VAR_INPUT
	WatchDog	: BOOL;
	// I/O Inputs 
		//FROM ENEDIS
		IN_CmdAutCpl_IO							: BOOL; 			(* Coupling Authorization (Autorisation de couplage)			              	*)
		IN_CmdAutCpl_End_IO						: BOOL; 			(* End of coupling Authorization (Fin d'autorisation de couplage)			    *)
		IN_CmdDisconnect_End_IO					: BOOL; 			(* End of disconnect order(Fin de demande de decouplage)                        *)
		IN_CmdDisconnect_IO						: BOOL;				(* Disconnect order(Demande de decouplage)                                      *)
		IN_CmdRSEOn_IO							: BOOL;				(* Start of RSE (Mise en RSE)                                                   *)
		IN_CmdRSEOff_IO							: BOOL;				(* Stop of RSE (Mise Hors RSE)                                                  *)
		IN_CmdStopPReg_IO						: BOOL;				(* Desactivation of P0 regulation(Fin de passage a P0)                          *)
		IN_CmdStartPReg_IO						: BOOL;				(* Activation of P0 regulation (Passage a P0)                                   *)
		IN_CmdStopQReg_IO						: BOOL;				(* Desactivation of Q0 regulation(Fin de passage a Q0)                          *)
		IN_CmdStartQreg_IO						: BOOL;				(* Activation of Q0 regulation(Passage a Q0)                                    *)
		IN_CmdEmergencyDisconnect_End_IO		: BOOL;				(* End of Emergency disconnect order(Fin demande d'effacement d'urgence) 	   	*)
		IN_CmdEmergencyDisconnect_IO			: BOOL;				(* Emergency disconnect order(Demande d'effacement d'urgence)                   *)
		IN_CmdDisconnectFromTac_IO				: BOOL; 			(* Teleaction disconnect(Decouplage par tac)                                    *)
		IN_CmdSynchro_IO						: BOOL;				(* Synchronisation signal														*)
		
		(* 4..20mA *)                                   			
		IN_MesP0Reg_IO							: INT; 				(* (kW)   Grid P0	*)
		IN_MesQ0Reg_IO							: INT; 				(* (KVar) Grid Q0 	*)
		IN_MesU0Reg_IO							: INT; 				(* (KV)   Grid V0   *)
		                                                			                                  			
		//FROM AKSES                                    			
		IN_CmdAutCpl_other						: BOOL; 			
		IN_CmdEmergencyDisconnect_other			: BOOL; 			
		IN_CmdEmergencyDisconnect_End_other		: BOOL; 			
		IN_CmdDisconnect_other					: BOOL; 			
		IN_CmdDisconnect_end_other				: BOOL; 			
		IN_CmdStartPReg_other					: BOOL; 			
		IN_CmdStartQReg_other					: BOOL; 			
		IN_CmdStopPReg_other					: BOOL; 			
		IN_CmdStopQReg_other					: BOOL;

		//FROM TAC 
		IN_CmdTAOn_IO							: BOOL; 			(* Teleaction in service(Teleaction en service)                                 *)
		IN_CmdTAOff_IO							: BOOL; 			(* Teleaction out of service (Teleaction Hors service)                          *)
		IN_CmdTacInFault_IO						: BOOL; 			(* Teleaction in fault(Défaut Tac)							 					*)
		IN_CmdOpenTAC_IO						: BOOL; 
		IN_CmdConsignationTAC_IO				: BOOL; 
		IN_CmdUnavailableTAC					: BOOL; 
			
		                                                			
		(*TC Relais Protection*)                        			
		IN_ConnectAuthorizationLost				: BOOL; 			// Tous les cas pour un Reset aut Couplage recu
		IN_Unavailable							: BOOL; 			// Disjoncteur général en Local, ou tous les départs en Local ou Bouton d'arret d'urgence 
		IN_PP_Connected							: BOOL; 			// Centrale Couplée si DG = Fermé et au moins 1 départ antenne en production et au moins un onduleur en Prod
                                     			
		OUT_MesFaultDecoupling_IO				: BOOL; 			(* Decoupling due to faults c13100 and c15400 combined with CB position    	*)
                                             			
END_VAR                                                 			
                                                        			
                                                        			
VAR_OUTPUT 

	// DEIE                                              			
		OUT_MesPPUnavailable_IO					: BOOL; 			(* TS centrale indisponible                                                	*)
		OUT_MesPPConnected_IO					: BOOL; 			(* Centrale couplée(1)/Centrale Découplée(0)                               	*)
		OUT_MesPPDisconnected_IO				: BOOL; 			(* Centrale Découplée														*)
		OUT_MesAutCpl_IO 						: BOOL; 			(* Autorisation de couplage reçue(1)/Attente d'autorisation de couplage(0)	*)
		OUT_MesAutCpl_end_IO 					: BOOL; 			(* Autorisation de couplage attente                                        	*)
		OUT_MesDisconnect_IO 					: BOOL; 			(* Demande de découplage reçue(1)/Fin de demande de découplage(0)         	*)
		OUT_MesDisconnect_End_IO 				: BOOL; 			(* Demande de découplage attente                                           	*)
		OUT_MesEmergencyDisconnect_IO 			: BOOL; 			(* Demande d effacement d'urgence reçue                                   	*)
		OUT_MesEmergencyDisconnect_End_IO 		: BOOL; 			(* Demande d effacement d'urgence attente		                          	*)
		OUT_MesRSEON_IO							: BOOL; 			(* Demande mise en RSE reçue                                              	*)
		OUT_MesRSEOff_IO						: BOOL; 			(* Demande mise en RSE en attente                                         	*)
		OUT_MesStartPReg_IO						: BOOL; 			(* Demande mise en regulation de P reçue                                  	*)
		OUT_MesStopPReg_IO						: BOOL; 			(* Demande mise en regulation de P en attente                             	*)
		OUT_MesStartQReg_IO						: BOOL; 			(* Demande mise en regulation de Q reçue                                  	*)
		OUT_MesStopQReg_IO						: BOOL; 			(* Demande mise en regulation de Q en attente	                          	*)
		
		(* 4..20mA *)                                   			
		OUT_MesP_IO							: REAL; 				(* (kW)   Grid P0	*)
		OUT_MesQ_IO							: REAL; 				(* (KVar) Grid Q0 	*)
		OUT_MesU_IO							: REAL; 				(* (KV)   Grid V0   *)
		
	// Synchro temporelle - EMS 
		Ecart_HeureGrid						: DINT;
		
	// TAC
		OUT_CmdTacInFault_IO					: BOOL; 
		OUT_MesOpenTAC_IO 						: BOOL; 
		OUT_MesTAOn_IO							: BOOL; 			(* Demande mise en TeleAction reçue                                       	*)
		OUT_MesTAOff_IO							: BOOL; 			(* Demande mise en TeleAction en attente                                  	*)
		
				
	// SOFREL
		
		OUT_MesP_IO_SOFREL					: REAL; 				(* (kW)   Grid P0	*)
		OUT_MesQ_IO_SOFREL					: REAL; 				(* (KVar) Grid Q0 	*)
		OUT_MesU_IO_SOFREL					: REAL; 				(* (KV)   Grid V0   *)
END_VAR


VAR PERSISTENT
	
END_VAR
VAR
		//TON
		TONConnectAuthorization					: TON;
		TONConnectAuthorization_end				: TON;
		TONEmergencyDisconnect	               	: TON;
	    TONEmergencyDisconnect_end	            : TON;
	    TONDisconnect	                		: TON;
	    TONDisconnect_end                		: TON;
	    TONPRegOn				                : TON;
	    TONPRegOff				                : TON;
	    TONQregOn				                : TON;
	    TONQRegOff				                : TON;
	    TONRSEOn				                : TON;
	    TONRSEOff				                : TON;
	    TONTAOn					                : TON;
	    TONTAOff				                : TON;
	
		R_Trig_SynchTime						: R_TRIG;

		Reste 									: DINT;
		Modulo 									: DINT;
		Heure_Pulse 							: DINT;
		bTest 									: BOOL;
END_VAR

METHOD M_AlarmManagement
//////////////////
// alarm and warning management
/////////////////

VAR 
	FB_AlarmCodeManager			: FB_AlarmCodeManager ; 
	
END_VAR
// ALARM CODE //
	FB_AlarmCodeManager(
		bAlarm1			:=MesDataExd.MesData.OUT_MesPPUnavailable, // Power plant is unavailable
		bAlarm2			:=FALSE, //
		bAlarm3			:=FALSE, //
		bAlarm4			:=FALSE, //
		bAlarm5			:=FALSE, //
		bAlarm6			:=FALSE, //
		bAlarm7			:=FALSE, //
		bAlarm8			:=FALSE, //
		bAlarm9			:=FALSE, //
		bAlarm10		:=FALSE, //
		bAlarm11		:=FALSE, //
		bAlarm12		:=FALSE, //
		bAlarm13		:=FALSE, //
		bAlarm14		:=FALSE, //
		bAlarm15		:=FALSE, //						 
		wAlarmCode		=>MesDataExd.MesData.MesAlarmCode);

// WARNING CODE //
	FB_AlarmCodeManager(		
		bAlarm1			:=IN_ConnectAuthorizationLost, 							//Loss of coupling authorization
		bAlarm2			:=FALSE,													//			
		bAlarm3			:=MesDataExd.MesData.OUT_SetptP > ParamPmaxPark OR MesDataExd.MesData.OUT_SetptP <= 0 ,		// P Setpoint from grid outside of permitted range
		bAlarm4			:=MesDataExd.MesData.OUT_SetptQ > ParamQMax OR MesDataExd.MesData.OUT_SetptQ <= ParamQMin, 	// Q Setpoint from grid outside of permitted range
		bAlarm5			:=MesDataExd.MesData.OUT_MesPPConnected						, 	//Powerplant is connected  
		bAlarm6			:=NOT MesDataExd.MesData.OUT_MesPPConnected					, 	//Powerplant is disconnected
		bAlarm7			:=MesDataExd.OUT_CmdPReg							    , 	//Q regulation mode is active     
		bAlarm8			:=NOT MesDataExd.MesData.OUT_CmdAutCpl		    		, 	//Waiting for coupling authorization	
		bAlarm9			:=MesDataExd.MesData.OUT_CmdDisconnect				, 	//Disconnect order
		bAlarm10		:=MesDataExd.MesData.OUT_CmdEmergencyDisconnect 	        , 	//Emergency Disconnect order
		bAlarm11		:=MesDataExd.OUT_CmdPReg												, 	// P regulation mode is active
		bAlarm12		:=MesDataExd.OUT_Rse								    , 	// RSE mode active  
		bAlarm13		:=MesDataExd.OUT_TA 							, 	//Teleaction active
		bAlarm14		:=IN_CmdDisconnectFromTac_IO , 		// Disconnect order from TAC
		bAlarm15		:=IN_CmdTacInFault_IO , 			// TAC in Fault 
		wAlarmCode		=>MesDataExd.MesData.MesWarningCode);		

// EVENT CODE 1//
	FB_AlarmCodeManager(
		bAlarm1			:=FALSE , // 
		bAlarm2			:=NOT MesDataExd.OUT_CmdPReg							    , 	//P regulation mode is inactive
		bAlarm3			:=MesDataExd.MesData.OUT_CmdAutCpl					, 	//Coupling authorization
		bAlarm4			:=FALSE ,//
		bAlarm5			:=IN_CmdSynchro_IO			    						, 	// Synchronization signal 
		bAlarm6			:=NOT MesDataExd.MesData.OUT_CmdDisconnect			, 	//End of disconnect order 
		bAlarm7			:=FALSE ,// 
		bAlarm8			:=NOT MesDataExd.MesData.OUT_CmdEmergencyDisconnect					, 	//End of Emergency Disconnect order
		bAlarm9			:=FALSE , // 
		bAlarm10		:=FALSE , // 
		bAlarm11		:=NOT MesDataExd.OUT_CmdPReg												, 	//P regulation mode is inactive
		bAlarm12		:=FALSE ,//  
		bAlarm13		:=NOT MesDataExd.OUT_Rse							    , 	//RSE mode inactive  
		bAlarm14		:=FALSE ,//
		bAlarm15		:=NOT MesDataExd.OUT_TA							, 	//Teleaction inactive
		wAlarmCode		=>MesDataExd.MesData.MesEventCode);   
                          	
// EVENT CODE 2 //		                                              	
	FB_AlarmCodeManager(                                              	
		bAlarm1			:=IN_CmdAutCpl_IO , 							// Coupling authorization received from DEIE
		bAlarm2			:=IN_CmdDisconnect_End_IO,						// End of disconnect order received from  DEIE
		bAlarm3			:=IN_CmdDisconnect_IO		   , 				// Disconnect order received from DEIE
		bAlarm4			:= IN_CmdEmergencyDisconnect_End_IO	   	, 		// End of Emergency disconnect order received from DEIE
		bAlarm5			:=IN_CmdAutCpl_other, 							// Coupling authoriztion received from HMI
		bAlarm6			:=IN_CmdDisconnect_other		 , 				// Disconnect order received from HMI
		bAlarm7			:=IN_CmdDisconnect_end_other,	 				// End of disconnect order received from HMI
		bAlarm8			:=IN_CmdEmergencyDisconnect_IO	, 				// Emergency disconnect order received from DEIE
		bAlarm9			:=IN_Unavailable, 								// Power plant is unavaiblable ( MainMVCB in local or ES) 
		bAlarm10		:=IN_CmdEmergencyDisconnect_other, 	//Emergency disconnect order received from HMI
		bAlarm11		:=IN_CmdEmergencyDisconnect_End_other	, 	//End of Emergency disconnect order received from HMI
		bAlarm12		:=FALSE, 	//
		bAlarm13		:=FALSE, 	//       
		bAlarm14		:=FALSE, 	//
		bAlarm15		:=FALSE	,//
		wAlarmCode		=>MesDataExd.MesData.MesEventCode2);
END_METHOD

METHOD M_CP
//////////////////
//  Emulator
/////////////////

VAR 
	// Method local variables (reinitialized at each cycle) 
	
END_VAR
END_METHOD

METHOD M_Evaluate
//////////////////
//  Evaluate grid variables 
/////////////////
VAR 
	// Method local variables (reinitialized at each cycle) 
	WatchDog	: BOOL;
END_VAR
WatchDog		:= TRUE;

//Filtering Input
	TONConnectAuthorization		(IN:=IN_CmdAutCpl_IO,PT:=ParamTONFiltering);
	TONEmergencyDisconnect		(IN:=IN_CmdEmergencyDisconnect_IO,PT:=ParamTONFiltering);	
	TONEmergencyDisconnect_end	(IN:=IN_CmdEmergencyDisconnect_End_IO,PT:=ParamTONFiltering);	
	TONDisconnect				(IN:=IN_CmdDisconnect_IO,PT:=ParamTONFiltering);	
	TONDisconnect_end			(IN:=IN_CmdDisconnect_End_IO,PT:=ParamTONFiltering);
	TONPRegOn				(IN:=IN_CmdStartPReg_IO,PT:=ParamTONFiltering);			
	TONPRegOff				(IN:=IN_CmdStopPReg_IO,PT:=ParamTONFiltering);				
	TONQregOn				(IN:=IN_CmdStartQreg_IO,PT:=ParamTONFiltering);				
	TONQRegOff				(IN:=IN_CmdStopQReg_IO,PT:=ParamTONFiltering);				
	TONRSEOn				(IN:=IN_CmdRSEOn_IO,PT:=ParamTONFiltering);				
	TONRSEOff				(IN:=IN_CmdRSEOff_IO,PT:=ParamTONFiltering);				
	TONTAOn					(IN:=IN_CmdTAOn_IO,PT:=ParamTONFiltering);					
	TONTAOff				(IN:=IN_CmdTAOff_IO,PT:=ParamTONFiltering);		

//Filtering Input
	TONConnectAuthorization		(IN:=IN_CmdAutCpl_IO,PT:=ParamTONFiltering);
	TONEmergencyDisconnect		(IN:=IN_CmdEmergencyDisconnect_IO,PT:=ParamTONFiltering);	
	TONEmergencyDisconnect_end	(IN:=IN_CmdEmergencyDisconnect_End_IO,PT:=ParamTONFiltering);	
	TONDisconnect				(IN:=IN_CmdDisconnect_IO,PT:=ParamTONFiltering);	
	TONDisconnect_end			(IN:=IN_CmdDisconnect_End_IO,PT:=ParamTONFiltering);
	TONPRegOn					(IN:=IN_CmdStartPReg_IO,PT:=ParamTONFiltering);			
	TONPRegOff					(IN:=IN_CmdStopPReg_IO,PT:=ParamTONFiltering);				
	TONQregOn					(IN:=IN_CmdStartQreg_IO,PT:=ParamTONFiltering);				
	TONQRegOff					(IN:=IN_CmdStopQReg_IO,PT:=ParamTONFiltering);				
	TONRSEOn					(IN:=IN_CmdRSEOn_IO,PT:=ParamTONFiltering);				
	TONRSEOff					(IN:=IN_CmdRSEOff_IO,PT:=ParamTONFiltering);				
	TONTAOn						(IN:=IN_CmdTAOn_IO,PT:=ParamTONFiltering);					
	TONTAOff					(IN:=IN_CmdTAOff_IO,PT:=ParamTONFiltering);	

// Calculate the difference between the closest hour and the trigger from GRID
	// closest hour is min betwenn the rest of the Euclydian division 3600s = 1h	
	R_Trig_SynchTime(CLK := IN_CmdSynchro_IO OR bTest);
	IF R_Trig_SynchTime.Q THEN
		Heure_Pulse	:= DT_TO_DINT(systemtime_to_dt(TIMESTR := CalLocalTimeStruct));
		Reste := Heure_Pulse MOD 3600;
		IF (3600-Reste) < Reste THEN
			Ecart_HeureGrid := -(3600-Reste);
		ELSE
			Ecart_HeureGrid := Reste;
		END_IF
		//Ecart_HeureGrid := MIN(3600-Reste, Reste);
		MesDataExd.MesEcart_HeureGrid := Ecart_HeureGrid;
	END_IF

//Converting P0 & Q0
	IF ParamP0Available THEN
		//OUT_P0 :=  (MesP0RegIO/ 32767.0) * REAL_TO_INT(ParamPmaxPark);
	MesDataExd.MesData.OUT_SetptP :=  (IN_MesP0Reg_IO/ 32767.0) * ABS(ParamPMin - ParamPmaxPark) + (ParamPMin);
	END_IF
	IF ParamQ0Available THEN
	MesDataExd.MesData.OUT_SetptQ := ( IN_MesQ0Reg_IO / 32767.0) * ABS(ParamQMin - ParamQMax) + (ParamQMin);
	END_IF	
//Logical Equation
	(*PLCUnavailable Si Watchdog n'est pas mis a jour a chaque temps de cycle Ou que la centrale est en Local *)
	MesDataExd.MesData.OUT_MesPPUnavailable := NOT WatchDog OR IN_Unavailable;
	
	(*Centrale Couplée *)
	MesDataExd.MesData.OUT_MesPPConnected := IN_PP_Connected;
	
	(*Autorisation de couplage*)
		IF TONConnectAuthorization.Q OR IN_CmdAutCpl_other THEN
		MesDataExd.MesData.OUT_CmdAutCpl := 1 ;
		END_IF
		
	(*Défaut GTE > 50s : Reset Aut Couplage recus*)
	(*Défaut C13_100 : Reset Aut Couplage recus*)
		IF IN_ConnectAuthorizationLost THEN  //IN_Long_GTE_Fault OR IN_C13_100_Fault OR IN_UnknownFault OR IN_3GTE_Fault THEN
		MesDataExd.MesData.OUT_CmdAutCpl  := FALSE ;
		END_IF
	
	(* RESEAU 6 ET 7 - DEMANDE DE DECOUPLAGE*)
		IF TONDisconnect.Q OR IN_CmdDisconnect_other THEN
			MesDataExd.MesData.OUT_CmdDisconnect := 1 ;
		END_IF
	
		IF TONDisconnect_end.Q OR IN_CmdDisconnect_end_other THEN
		MesDataExd.MesData.OUT_CmdDisconnect := 0 ;
		END_IF

	(* RESEAU 8 ET 9 - DEMANDE D’EFFACEMENT D’URGENCE*)
		IF TONEmergencyDisconnect.Q OR  IN_CmdEmergencyDisconnect_other THEN
		MesDataExd.MesData.OUT_CmdEmergencyDisconnect := 1 ;
		END_IF
	
		IF TONEmergencyDisconnect_end.Q OR IN_CmdEmergencyDisconnect_End_other THEN
		MesDataExd.MesData.OUT_CmdEmergencyDisconnect := 0 ;
		END_IF
	(* RESEAU 10 ET 11 - PASSAGE A P0*)
		IF TONPRegOn.Q OR IN_CmdStartPReg_other THEN
		MesDataExd.OUT_CmdPReg := 1 ;
		END_IF
		
		IF TONPRegOff.Q OR IN_CmdStopPReg_other THEN
		MesDataExd.OUT_CmdPReg := 0 ;
		END_IF
		
	(* RESEAU 12 ET 13 - PASSAGE A Q0*)
		IF TONQregOn.Q OR IN_CmdStartQReg_other THEN
		MesDataExd.OUT_CmdQReg := 1 ;
		END_IF
		
		IF TONQregOff.Q OR IN_CmdStopQReg_other THEN
		MesDataExd.OUT_CmdQReg := 0 ;
		END_IF

				
	(* RSE*)
		IF TONRSEOn.Q  THEN
		MesDataExd.OUT_Rse := 1 ;
		ELSIF TONRSEOff.Q THEN
		MesDataExd.OUT_Rse := 0 ;
		END_IF
		
	(* TA*)
		IF TONTAOn.Q  THEN
		MesDataExd.OUT_TA := 1 ;
		ELSIF TONTAOff.Q THEN
		MesDataExd.OUT_TA := 0 ;
		END_IF
		
	
// Update Outputs IO to GRID 
OUT_MesPPUnavailable_IO				:= MesDataExd.MesData.OUT_MesPPUnavailable ; 			
OUT_MesPPConnected_IO				:= MesDataExd.MesData.OUT_MesPPConnected ; 	
OUT_MesPPDisconnected_IO			:= NOT MesDataExd.MesData.OUT_MesPPConnected ; 
OUT_MesAutCpl_IO 					:= MesDataExd.MesData.OUT_CmdAutCpl ; 			
OUT_MesAutCpl_end_IO 				:= NOT MesDataExd.MesData.OUT_CmdAutCpl ; 		
OUT_MesDisconnect_IO 				:= MesDataExd.MesData.OUT_CmdDisconnect ; 		
OUT_MesDisconnect_End_IO 			:= NOT MesDataExd.MesData.OUT_CmdDisconnect ; 		
OUT_MesEmergencyDisconnect_IO 		:= MesDataExd.MesData.OUT_CmdEmergencyDisconnect ; 		
OUT_MesEmergencyDisconnect_End_IO 	:= NOT MesDataExd.MesData.OUT_CmdEmergencyDisconnect ; 		

OUT_MesRSEON_IO						:= MesDataExd.OUT_Rse ;
OUT_MesRSEOff_IO					:= NOT MesDataExd.OUT_Rse ;
OUT_MesTAOn_IO						:= MesDataExd.OUT_TA ; 
OUT_MesTAOff_IO						:= NOT MesDataExd.OUT_TA ; 

OUT_MesStartPReg_IO	 := MesDataExd.OUT_CmdPReg ; 
OUT_MesStopPReg_IO	 := NOT MesDataExd.OUT_CmdPReg ; 
OUT_MesStartQReg_IO	 := MesDataExd.OUT_CmdQReg ; 
OUT_MesStopQReg_IO	 := NOT MesDataExd.OUT_CmdQReg ;
END_METHOD

METHOD M_Execute
//////////////////
//  Method Calls 
/////////////////
VAR 
	// Method local variables (reinitialized at each cycle) 
	
END_VAR
// PERMANENT CONDITIONS //
	M_CP() ; 
	
// METHODS CALLS //
	IF bInit THEN
		M_Init() ; 
		bInit:= FALSE ; 
	ELSIF CmdInit_G THEN 
		bInit:= TRUE ;
	END_IF

	M_Evaluate() ; 
	M_AlarmManagement();
END_METHOD

METHOD M_Init
VAR 

END_VAR
// Au démarrage du code , on maintient en mémoire l'autorization de couplage ssi la centrale est connectée. 
IF NOT A1_SUBMV.A1_MainMVCB.MesDataExd.MesData.MesClosed THEN // La centrale n'est pas connectée
	MesDataExd.MesData.OUT_CmdAutCpl := FALSE ;
	MesDataExd.OUT_CmdPReg := FALSE;
	MesDataExd.OUT_CmdQReg := FALSE;

END_IF
END_METHOD

END_FUNCTION_BLOCK

// ---- 01_Equipement_Library/GRID/FB_GRID_PLAN.TcPOU
FUNCTION_BLOCK FB_GRID_PLAN
//////////////////
// Grid Operator interface . Base FB
//////////////////
VAR_INPUT PERSISTENT
	// Parameters of the Object (instance specific) 
		ParamRseAvailable						: BOOL:=TRUE		; // GRID with RSE option
		ParamTaAvailable						: BOOL:=TRUE		; // GRID with Teleaction option
		ParamP0Available						: BOOL:=TRUE		; // GRID with P regulation option
		ParamQ0Available						: BOOL:=TRUE		; // GRID with Q regulation option
		ParamTONFiltering						: TIME:=T#200MS		; // Minimum tempo filter before command validation (Noise filtering)
		ParamPmaxPark							: REAL;					//(kW) Contractual maximal power plant active power
		ParamQMax								: REAL;					// (Kvar)   Contractual maximal power plant reactive power
		ParamQMin								: REAL; 				// (Kvar)  Contractual maximal power plant reactive power
		ParamPMin								: REAL;					// (kW) Contractual minimal power plant active power
		
		
		MesDataExd							AT%Q* 		: GRID_PLAN;	
		
END_VAR


VAR_INPUT
	// I/O Inputs 
		//FROM ENEDIS
		IN_CmdAutCpl_IO								: BOOL; //Autorisation de couplage
		IN_CmdDisconnect_End_IO						: BOOL; //Fin de demande de decouplage
		IN_CmdDisconnect_IO							: BOOL;	//Demande de decouplage
		IN_CmdRSEOn_IO								: BOOL;	//Mise en RSE
		IN_CmdRSEOff_IO								: BOOL;	//Mise Hors RSE
		IN_CmdTAOn_IO								: BOOL; //Teleaction en service
		IN_CmdTAOff_IO								: BOOL; //Teleaction Hors service
		IN_CmdStopPReg_IO							: BOOL;	//Fin de passage a P0
		IN_CmdStartPReg_IO							: BOOL;	//Passage a P0
		IN_CmdStopQReg_IO							: BOOL;	//Fin de passage a Q0
		IN_CmdStartQreg_IO							: BOOL;	//Passage a Q0
		IN_CmdEndDisconnectOrder_IO					: BOOL;	//Fin demande d'effacement d'urgence		
		IN_CmdEmergencyDisconnect_IO				: BOOL;	//Demande d'effacement d'urgence
		IN_CmdDisconnectFromTac_IO					: BOOL; //Decouplage par tac
		IN_CmdTacInFault_IO							: BOOL; //Défaut Tac
		(* 4..20mA *)
		IN_MesP0Reg_IO								: INT; //Kw
		IN_MesQ0Reg_IO								: INT; //Kvar
		
		
		//FROM AKSES
		IN_CmdAutCpl_other							: BOOL;
		IN_CmdEmergencyDisconnect_other				: BOOL;
		IN_CmdEmergencyDisconnect_End_other			: BOOL;
		IN_CmdDisconnect_other						: BOOL;
		IN_CmdDisconnect_end_other					: BOOL;
		IN_CmdStartPReg_other						: BOOL;
		IN_CmdStartQReg_other						: BOOL;
		IN_CmdStopPReg_other						: BOOL;
		IN_CmdStopQReg_other						: BOOL;
		
		IN_SetptP_other								: REAL;
		IN_SetptQ_other								: REAL;
		IN_SetptPF_other							: REAL;
		IN_SetptU_other								: REAL;
		
		(*TC Relais Protection*)
		IN_ConnectAuthorizationLost				: BOOL; (*Tous les cas pour un Reset aut Couplage recu*)
		IN_Unavailable							: BOOL; (*Disjoncteur général en Local, ou tous les départs en Local ou Bouton d'arret d'urgence *)
		IN_PP_Connected							: BOOL; (*Centrale Couplée si DG = Fermé et au moins 1 départ antenne en production et au moins un onduleur en Prod*)
	    IN_CmdToggleRead						: BOOL;	

END_VAR 


VAR_OUTPUT
		OUT_MesPPUnavailable_IO					: BOOL; (*TS centrale indisponible*)
		OUT_MesPPConnected_IO					: BOOL; (*Centrale couplée(1)/Centrale Découplée(0)*)
		OUT_MesAutCpl_IO 						: BOOL; (*Autorisation de couplage reçue(1)/Attente d'autorisation de couplage(0)*)
		OUT_MesAutCpl_end_IO 						: BOOL; (*Autorisation de couplage attente*)
		OUT_MesDisconnect_IO 					: BOOL; (*Demande de découplage reçue(1)/Fin de demande de découplage(0)*)
		OUT_MesDisconnect_End_IO 					: BOOL; (*Demande de découplage attente*)		
		OUT_MesEmergencyDisconnect_IO 			: BOOL; (*Demande d effacement d'urgence reçue*)
		OUT_MesEmergencyDisconnect_End_IO 			: BOOL; (*Demande d effacement d'urgence attente*)		
END_VAR



VAR
	//M_ALARMMANAGEMENT VARIABLES//                                                    								


	//M_EVALUATE VARIABLES//
		//

		//TON
		TONConnectAuthorization					: TON;
		TONEmergencyDisconnect	               	: TON;
	    TONEmergencyDisconnect_end	            : TON;
	    TONDisconnect	                		: TON;
	    TONDisconnect_end                		: TON;
	    TONPRegOn				                : TON;
	    TONPRegOff				                : TON;
	    TONQregOn				                : TON;
	    TONQRegOff				                : TON;
	    TONRSEOn				                : TON;
	    TONRSEOff				                : TON;
	    TONTAOn					                : TON;
	    TONTAOff				                : TON;
		
	//M_Evaluate
	// IEC 104
		MesDataIEC						: IEC104_PLAN;
		AODB 							: ARRAY[0..GVL_Cst.CstNbAOEntries] OF ST_IEC870_5_101AODBEntry ;
		memory 			AT%MB0			: ARRAY[0..200] OF BYTE;
		FB_IEC							: FB_IEC104ServerAkuo;(* Controlled station function block instance *)

	
	//M_INIT VARIABLES //
		bInit					: BOOL:= TRUE;	
		initError				: UDINT;
		bBoot					: BOOL := TRUE ;		// Boolean that indicates a restart of the PLC .
	// M_EXECUTE VARIABLES //
        Trig_Cmd_Read			: R_TRIG;                                                                                        
		
		   		                    		
        SetptP_IEC_Old 			: REAL;
		SetptQ_IEC_Old 			: REAL;
		SetptU_IEC_Old 			: REAL;
		SetptCosPhi_IEC_Old 	: REAL;
		
		bChange_SetptP_IEC 		: BOOL;
		bChange_SetptQ_IEC 		: BOOL;
		bChange_SetptU_IEC 		: BOOL;
		bChange_SetptCosPhi_IEC	: BOOL;

		   		                    		
        SetptP_Manu_Old 		: REAL;
		SetptQ_Manu_Old 		: REAL;
		SetptU_Manu_Old 		: REAL;
		SetptCosPhi_Manu_Old	: REAL;
				     
		bChange_SetptP_Manu		: BOOL;
		bChange_SetptQ_Manu		: BOOL;
		bChange_SetptU_Manu		: BOOL;
		bChange_SetptCosPhi_Manu: BOOL;
		
		
        CmdQ_Old				: REAL;             
		bChange_CmdQ_Old		: BOOL;
				
END_VAR

METHOD M_AlarmManagement
//////////////////
// alarm and warning management
/////////////////

VAR 
	FB_AlarmCodeManager			: FB_AlarmCodeManager ; 
	
END_VAR
// ALARM CODE //
	FB_AlarmCodeManager(
		bAlarm1			:=MesDataExd.mesData.OUT_MesPPUnavailable, // Power plant is unavailable
		bAlarm2			:=FALSE , //
		bAlarm3			:=FALSE, //
		bAlarm4			:=FALSE, //
		bAlarm5			:=FALSE, //
		bAlarm6			:=FALSE, //
		bAlarm7			:=FALSE, //
		bAlarm8			:=FALSE, //
		bAlarm9			:=FALSE, //
		bAlarm10		:=FALSE, //
		bAlarm11		:=FALSE, //
		bAlarm12		:=FALSE, //
		bAlarm13		:=FALSE, //
		bAlarm14		:=FALSE, //
		bAlarm15		:=FALSE, //						 
		wAlarmCode		=> MesDataExd.MesData.MesAlarmCode);

// WARNING CODE //
	FB_AlarmCodeManager(		
		bAlarm1			:=IN_ConnectAuthorizationLost, 							//Loss of coupliong authorization
		bAlarm2			:=FALSE,													//			
		bAlarm3			:=MesDataExd.MesData.OUT_SetptP > ParamPmaxPark OR MesDataExd.MesData.OUT_SetptP <= 0 ,		// P Setpoint from grid outside of permitted range
		bAlarm4			:=MesDataExd.MesData.OUT_SetptQ > ParamQMax OR MesDataExd.MesData.OUT_SetptQ <= ParamQMin, 	// Q Setpoint from grid outside of permitted range
		bAlarm5			:=MesDataExd.MesData.OUT_MesPPConnected						, 	//Powerplant is connected  
		bAlarm6			:=NOT MesDataExd.MesData.OUT_MesPPConnected					, 	//Powerplant is disconnected
		bAlarm7			:=FB_IEC.eComState = INIT,  // IEC server is Initializing
		bAlarm8			:=FB_IEC.eComState = IDLE,  // ieC server is Idle
		bAlarm9			:=FALSE,  //
		bAlarm10		:=FALSE,  //
		bAlarm11		:=FALSE,  //
		bAlarm12		:=FALSE,  //
		bAlarm13		:=FALSE,  //
		bAlarm14		:=FALSE,  //
		bAlarm15		:=FALSE  , // 
		wAlarmCode		=> MesDataExd.MesData.MesWarningCode);		

// EVENT CODE 1//
	FB_AlarmCodeManager(
		bAlarm1			:=FALSE , // 
		bAlarm2			:=FALSE , // A1_PP.IN_CmdQ=0,
		bAlarm3			:=bChange_SetptU_Manu,								// Change on U control mode
		bAlarm4			:=bChange_CmdQ_Old, 								// Change on Q control mode	
		bAlarm5			:=bChange_SetptCosPhi_IEC, 							// Change of PF setpoint from IEC
		bAlarm6			:=bChange_SetptCosPhi_Manu, 						// Change of PF setpoint from HMI
		bAlarm7			:=MesDataExd.MEsData.OUT_CmdDisconnect, 			// Disconnect order
		bAlarm8			:=bChange_SetptP_Manu,								// Change of P setpoint from HMI
		bAlarm9			:=bChange_SetptQ_IEC,								// Change of Q setpoint from IEC
		bAlarm10		:=FALSE , // A1_PP.IN_CmdQ=1,									// Control mode is in QvU mode
		bAlarm11		:=FALSE , // A1_PP.IN_CmdQ=2,									// Control mode is in PF mode
		bAlarm12		:=FALSE , // A1_PP.IN_CmdQ=3,									// Control mode is in Q mode 
		bAlarm13		:=FALSE , // A1_PP.IN_CmdQ=4,									// Control mode is in U mode
		bAlarm14		:=bChange_SetptQ_Manu,								// Change of Q setpoint from HMI
		bAlarm15		:=bChange_SetptU_IEC,								// Change of U setpoint from IEC
		wAlarmCode		=> MesDataExd.MesData.MesEventCode);   
                          	
// EVENT CODE 2 //		                                              	
	FB_AlarmCodeManager(                                              	
		bAlarm1			:=FALSE , //
		bAlarm2			:=FALSE , //
		bAlarm3			:=FALSE, 	//
		bAlarm4			:=FALSE	, 	//
		bAlarm5			:=FALSE, 	//
		bAlarm6			:=FALSE, 	//
		bAlarm7			:=FALSE, 	//
		bAlarm8			:=FALSE	, 	// 
		bAlarm9			:=FALSE, 	//
		bAlarm10		:=FALSE, 	//
		bAlarm11		:=FALSE	, 	//
		bAlarm12		:=FALSE, 	//
		bAlarm13		:=FALSE, 	//       
		bAlarm14		:=FALSE, 	//
		bAlarm15		:=FALSE	,//
		wAlarmCode		=> MesDataExd.MesData.MesEventCode2);
END_METHOD

METHOD M_CP
//////////////////
//  Emulator
/////////////////

VAR 
	// Method local variables (reinitialized at each cycle) 
	
END_VAR


SUPER^.M_CP() ; 




Trig_Cmd_Read(CLK:=IN_CmdToggleRead);
	
IF Trig_Cmd_Read.Q THEN
	IN_CmdToggleRead := FALSE;
	MesDataExd.MesData.MesCP_Read := NOT MesDataExd.MesData.MesCP_Read;
END_IF
END_METHOD

METHOD M_Evaluate
//////////////////
//  Read Modbus Variable for PCS . 
/////////////////
VAR 
	// Method local variables (reinitialized at each cycle) 
	WatchDog	: BOOL;
END_VAR
WatchDog		:= TRUE;



//Filtering Input
	TONConnectAuthorization		(IN:=IN_CmdAutCpl_IO,PT:=ParamTONFiltering);
	TONEmergencyDisconnect		(IN:=IN_CmdEmergencyDisconnect_IO,PT:=ParamTONFiltering);	
	TONEmergencyDisconnect_end	(IN:=IN_CmdEndDisconnectOrder_IO,PT:=ParamTONFiltering);	
	TONDisconnect				(IN:=IN_CmdDisconnect_IO,PT:=ParamTONFiltering);	
	TONDisconnect_end			(IN:=IN_CmdDisconnect_End_IO,PT:=ParamTONFiltering);
	TONPRegOn					(IN:=IN_CmdStartPReg_IO,PT:=ParamTONFiltering);			
	TONPRegOff					(IN:=IN_CmdStopPReg_IO,PT:=ParamTONFiltering);				
	TONQregOn					(IN:=IN_CmdStartQreg_IO,PT:=ParamTONFiltering);				
	TONQRegOff					(IN:=IN_CmdStopQReg_IO,PT:=ParamTONFiltering);				
	TONRSEOn					(IN:=IN_CmdRSEOn_IO,PT:=ParamTONFiltering);				
	TONRSEOff					(IN:=IN_CmdRSEOff_IO,PT:=ParamTONFiltering);				
	TONTAOn						(IN:=IN_CmdTAOn_IO,PT:=ParamTONFiltering);					
	TONTAOff					(IN:=IN_CmdTAOff_IO,PT:=ParamTONFiltering);		

////Converting P0 & Q0
//	IF ParamP0Available THEN
//		//MesData.OUT_P0 :=  (MesP0RegIO/ 32767.0) * REAL_TO_INT(ParamPmaxPark);
//		MesDataExd.MesData.OUT_SetptP :=  (IN_MesP0Reg_IO/ 32767.0) * ABS(ParamPMin - ParamPmaxPark) + (ParamPMin);
//	END_IF
//	IF ParamQ0Available THEN
//		MesDataExd.MesData.OUT_SetptQ := ( IN_MesQ0Reg_IO / 32767.0) * ABS(ParamQMin - ParamQMax) + (ParamQMin);
//	END_IF	
//Logical Equation
	(*PLCUnavailable Si Watchdog n'est pas mis a jour a chaque temps de cycle Ou que la centrale est en Local *)
		MesDataExd.MesData.OUT_MesPPUnavailable := NOT WatchDog OR IN_Unavailable;
	
	(*Centrale Couplée *)
		//MesDataExd.MesData.OUT_MesPPConnected := IN_PP_Connected;
	
	(*Autorisation de couplage*)
		IF TONConnectAuthorization.Q OR IN_CmdAutCpl_other THEN
			MesDataExd.MEsData.OUT_CmdAutCpl := 1 ;
		END_IF
		
	(*Défaut GTE > 50s : Reset Aut Couplage recus*)
	(*Défaut C13_100 : Reset Aut Couplage recus*)
		IF IN_ConnectAuthorizationLost THEN  //IN_Long_GTE_Fault OR IN_C13_100_Fault OR IN_UnknownFault OR IN_3GTE_Fault THEN
			MesDataExd.MEsData.OUT_CmdAutCpl  := FALSE ;
		END_IF
	
	(* RESEAU 6 ET 7 - DEMANDE DE DECOUPLAGE*)
		IF TONDisconnect.Q OR IN_CmdDisconnect_other THEN
			 MesDataExd.MEsData.OUT_CmdDisconnect := 1 ;
		END_IF
	
		IF TONDisconnect_end.Q OR IN_CmdDisconnect_end_other THEN
			MesDataExd.MEsData.OUT_CmdDisconnect := 0 ;
		END_IF

	(* RESEAU 8 ET 9 - DEMANDE D’EFFACEMENT D’URGENCE*)
		IF TONEmergencyDisconnect.Q OR  IN_CmdEmergencyDisconnect_other THEN
			MesDataExd.MEsData.OUT_CmdEmergencyDisconnect := 1 ;
		END_IF
	
		IF TONEmergencyDisconnect_end.Q OR IN_CmdEmergencyDisconnect_End_other THEN
			MesDataExd.MEsData.OUT_CmdEmergencyDisconnect := 0 ;
		END_IF
	(* RESEAU 10 ET 11 - PASSAGE A P0*)
		IF TONPRegOn.Q OR IN_CmdStartPReg_other THEN
			MesDataExd.OUT_CmdPReg := 1 ;
		END_IF
		
		IF TONPRegOff.Q OR IN_CmdStopPReg_other THEN
			MesDataExd.OUT_CmdPReg := 0 ;
		END_IF
		
	(* RESEAU 12 ET 13 - PASSAGE A Q0*)
		IF TONQregOn.Q OR IN_CmdStartQReg_other THEN
			MesDataExd.OUT_CmdQReg := 1 ;
		END_IF
		
		IF TONQregOff.Q OR IN_CmdStopQReg_other THEN
			MesDataExd.OUT_CmdQReg := 0 ;
		END_IF

				
	(* RSE*)
		IF TONRSEOn.Q  THEN
			MesDataExd.OUT_Rse := 1 ;
		ELSIF TONRSEOff.Q THEN
			MesDataExd.OUT_Rse := 0 ;
		END_IF
		
	(* TA*)
		IF TONTAOn.Q  THEN
			MesDataExd.OUT_TA := 1 ;
		ELSIF TONTAOff.Q THEN
			MesDataExd.OUT_TA := 0 ;
		END_IF
		

// Update Outputs IO to GRID 
OUT_MesPPUnavailable_IO				:= MEsDataExd.MesData.OUT_MesPPUnavailable ; 			
OUT_MesPPConnected_IO				:= MEsDataExd.MesData.OUT_MesPPConnected ; 				 
OUT_MesAutCpl_IO 					:= MEsDataExd.MesData.OUT_CmdAutCpl ; 			
OUT_MesAutCpl_end_IO 				:= NOT MEsDataExd.MesData.OUT_CmdAutCpl ; 		
OUT_MesDisconnect_IO 				:= MEsDataExd.MesData.OUT_CmdDisconnect ; 		
OUT_MesDisconnect_End_IO 			:= NOT MEsDataExd.MesData.OUT_CmdDisconnect ; 		
OUT_MesEmergencyDisconnect_IO 		:= MEsDataExd.MesData.OUT_CmdEmergencyDisconnect ; 		
OUT_MesEmergencyDisconnect_End_IO 	:= NOT MEsDataExd.MesData.OUT_CmdEmergencyDisconnect ; 		

// Values of IEC
	MesDataIEC.OUT_MesAvailability := A1_PP.MesData.MesPsol_Connected / (38*6);
	MesDataIEC.OUT_MesGHI := A1_WS.MesDataExd.Pyran_GHI.MesData.Value ;
	MesDataIEC.OUT_MesGTI := (A1_WS.MesDataExd.Pyran_GTI_PTR1_1.MesData.Value + A1_WS.MesDataExd.Pyran_GTI_PTR1_2.MesData.Value)/2;
	MesDataIEC.OUT_MesI_33kV_1	:= A1_SUBMV.A1_PM.MesDataExd.MesData.MesI1;
	MesDataIEC.OUT_MesI2_110kV	:= A1_SUBHV.A1_PM.MesDataExd.MesData.MesI2;
	MesDataIEC.OUT_MesI2_33kV	:= A1_SUBMV.A1_PM.MesDataExd.MesData.MesI2;
	MesDataIEC.OUT_MesP_110kV	:= A1_SUBHV.A1_PM.MesDataExd.MesData.MesP/1000;
	MesDataIEC.OUT_MesP_33kV	:= A1_SUBMV.A1_PM.MesDataExd.MesData.MesP/1000;
	MesDataIEC.OUT_MesP_33kV_1	:= A1_SUBMV.A1_PM.MesDataExd.MesData.MesP/1000;
	MesDataIEC.OUT_MesPMax		:= A1_PP.ParamPmax/1000;
	MesDataIEC.OUT_MesQ_110kV	:= A1_SUBHV.A1_PM.MesDataExd.MesData.MesQ/1000;
	MesDataIEC.OUT_MesQ_33kV	:= A1_SUBMV.A1_PM.MesDataExd.MesData.MesQ/1000;
	MesDataIEC.OUT_MesQ_33kV_1	:= A1_SUBMV.A1_PM.MesDataExd.MesData.MesQ/1000;
//	MesDataIEC.OUT_MesTempAmb	:= (A1_WS.MesDataExd.AX_Datalogger[1].TempSensor_Ext.Value + A1_WS.MesDataExd.AX_Datalogger[2].TempSensor_Ext.Value)/2;
	MesDataIEC.OUT_MesTempPan	:= (A1_WS.MesDataExd.TempSensor_Panel_PTR1.MesData.Value) ;
	MesDataIEC.OUT_MesU_33kV_1	:= A1_SUBMV.A1_PM.MesDataExd.MesData.MesU12/1000;
	MesDataIEC.OUT_MesU12_110kV	:= A1_SUBHV.A1_PM.MesDataExd.MesData.MesU12/1000;
	MesDataIEC.OUT_MesU12_33kV	:= A1_SUBMV.A1_PM.MesDataExd.MesData.MesU12/1000;


	
MesDataIEC.OUT_MesDouble.0 := MesDataIEC.OUT_MesPosCB_SubMV;
MesDataIEC.OUT_MesDouble.1 := NOT MesDataIEC.OUT_MesPosCB_SubMV;

MesDataIEC.OUT_MesDouble.2 := MesDataIEC.OUT_MesPosSec_SubMV;
MesDataIEC.OUT_MesDouble.3 := NOT MesDataIEC.OUT_MesPosSec_SubMV;

MesDataIEC.OUT_MesDouble.4 := MesDataIEC.OUT_MesPosEarth_SubMV;
MesDataIEC.OUT_MesDouble.5 := NOT MesDataIEC.OUT_MesPosEarth_SubMV;

MesDataIEC.OUT_MesDouble.6 := MesDataIEC.OUT_CmdPvF_On;
MesDataIEC.OUT_MesDouble.7 := NOT MesDataIEC.OUT_CmdPvF_On;

IF MesDataIEC.OUT_CmdP = 0 THEN
	MesDataIEC.OUT_MesDouble2.2 := TRUE; 
    MesDataIEC.OUT_MesDouble2.3 := FALSE;

ELSIF mesDataIEC.OUT_CmdP = 1 THEN
	MesDataIEC.OUT_MesDouble2.2 := FALSE;
    MesDataIEC.OUT_MesDouble2.3 := TRUE;
END_IF


IF MesDataIEC.OUT_CmdQ = 3 THEN
	MesDataIEC.OUT_MesDouble4.2 := FALSE;
	MesDataIEC.OUT_MesDouble4.3 := FALSE;
ELSIF mesDataIEC.OUT_CmdQ = 1 THEN
	MesDataIEC.OUT_MesDouble4.2 := TRUE; 
	MesDataIEC.OUT_MesDouble4.3 := FALSE;
ELSIF mesDataIEC.OUT_CmdQ = 2 THEN
	MesDataIEC.OUT_MesDouble4.2 := FALSE; 
	MesDataIEC.OUT_MesDouble4.3 := TRUE;
ELSIF mesDataIEC.OUT_CmdQ = 0 THEN
	MesDataIEC.OUT_MesDouble4.2 := TRUE; 
	MesDataIEC.OUT_MesDouble4.3 := TRUE;
END_IF




MesDataIEC.OUT_MesDouble2.4 := MesDataIEC.OUT_CmdQ_On;
MesDataIEC.OUT_MesDouble2.5 := NOT MesDataIEC.OUT_CmdQ_On;

MesDataIEC.OUT_MesDouble2.6 := MesDataIEC.OUT_MesPosInter_33kV;
MesDataIEC.OUT_MesDouble2.7 := NOT MesDataIEC.OUT_MesPosInter_33kV;

MesDataIEC.OUT_MesDouble3.0 := MesDataIEC.OUT_MesPosSecLinea_33kV;
MesDataIEC.OUT_MesDouble3.1 := NOT MesDataIEC.OUT_MesPosSecLinea_33kV;

MesDataIEC.OUT_MesDouble3.2 := MesDataIEC.OUT_MesPosSec_33kV;
MesDataIEC.OUT_MesDouble3.3 := NOT MesDataIEC.OUT_MesPosSec_33kV;

MesDataIEC.OUT_MesDouble3.4 := MesDataIEC.OUT_MesPosEarth_33kV;
MesDataIEC.OUT_MesDouble3.5 := NOT MesDataIEC.OUT_MesPosEarth_33kV;

MesDataIEC.OUT_MesDouble3.6 := MesDataIEC.OUT_MesPosInter_110kV;
MesDataIEC.OUT_MesDouble3.7 := NOT MesDataIEC.OUT_MesPosInter_110kV;

MesDataIEC.OUT_MesDouble4.0 := MesDataIEC.OUT_MesPosSecLinea_110kV;
MesDataIEC.OUT_MesDouble4.1 := NOT MesDataIEC.OUT_MesPosSecLinea_110kV;




// Writing commands
	// Grid command
		//IF SetptP_IEC_Old <> MesDataIEC.IN_SetptP THEN
		//	SetptP_IEC_Old := MesDataIEC.IN_SetptP;
		//	MesDataExd.MesData.OUT_SetptP := MesDataIEC.IN_SetptP;
		//END_IF

	// Grid command
		IF MesDataIEC.OUT_CmdQ_On AND SetptQ_IEC_Old <> MesDataIEC.IN_SetptQ THEN
			SetptQ_IEC_Old 							:= MesDataIEC.IN_SetptQ;
			MesDataExd.MesData.OUT_SetptQ 			:=MesDataIEC.IN_SetptQ*1000;
			A1_PP.IN_SetptQ							:= MesDataIEC.IN_SetptQ*1000;
			bChange_SetptQ_IEC						:= TRUE;
		ELSE
			bChange_SetptQ_IEC						:= FALSE;
		END_IF
	
		IF MesDataIEC.OUT_CmdQ_On AND SetptU_IEC_Old <> MesDataIEC.IN_SetptU THEN
			SetptU_IEC_Old 							:= MesDataIEC.IN_SetptU;
			MesDataExd.MesData.OUT_SetptU 			:= MesDataIEC.IN_SetptU*1000;
			A1_PP.IN_SetptU							:= MesDataIEC.IN_SetptU*1000;
			bChange_SetptU_IEC						:= TRUE;
		ELSE
			bChange_SetptU_IEC						:= FALSE;
		END_IF
		
		IF MesDataIEC.OUT_CmdQ_On AND SetptCosPhi_IEC_Old <> MesDataIEC.IN_SetptPF THEN
			SetptCosPhi_IEC_Old 					:= MesDataIEC.IN_SetptPF ;
			MesDataExd.MesData.OUT_SetptCosPhi 		:= MesDataIEC.IN_SetptPF;
			A1_PP.IN_SetptCosPhi					:= MesDataIEC.IN_SetptPF;
			bChange_SetptCosPhi_IEC					:= TRUE;
		ELSE
			bChange_SetptCosPhi_IEC					:= FALSE;
		END_IF
				

	// Manual command from OPCUA
		IF SetptP_Manu_Old <> IN_SetptP_other THEN
			SetptP_Manu_Old 						:= IN_SetptP_other ;
			MesDataExd.MesData.OUT_SetptP 			:= IN_SetptP_other;
			A1_PP.IN_SetptP 						:= IN_SetptP_other;
			bChange_SetptP_Manu						:= TRUE;
		ELSE
			bChange_SetptP_Manu						:= FALSE;
		END_IF
		
		IF SetptCosPhi_Manu_Old <> IN_SetptPF_other THEN
			SetptCosPhi_Manu_Old					:= IN_SetptPF_other ;
			MesDataExd.MesData.OUT_SetptCosPhi		:= IN_SetptPF_other;
			A1_PP.IN_SetptCosPhi					:= IN_SetptPF_other;
			bChange_SetptCosPhi_Manu				:= TRUE;
		ELSE
			bChange_SetptCosPhi_Manu				:= FALSE;
		END_IF
		
		IF SetptU_Manu_Old <> IN_SetptU_other THEN
			SetptU_Manu_Old 						:= IN_SetptU_other ;
			MesDataExd.MesData.OUT_SetptU 			:= IN_SetptU_other;
			A1_PP.IN_SetptU							:= IN_SetptU_other;
			bChange_SetptU_Manu						:= TRUE;
		ELSE
			bChange_SetptU_Manu						:= FALSE;
		END_IF

		IF SetptQ_Manu_Old <> IN_SetptQ_other THEN
			SetptQ_Manu_Old 						:= IN_SetptQ_other ;
			MesDataExd.MesData.OUT_SetptQ 			:= IN_SetptQ_other;
			A1_PP.IN_SetptQ							:= IN_SetptQ_other;
			bChange_SetptQ_Manu						:= TRUE;
		ELSE
			bChange_SetptQ_Manu						:= FALSE;
		END_IF
	
		
// Changing Q control mode 
	IF MesDataIEC.OUT_CmdQ_On AND  MesDataIEC.IN_CmdQ <> CmdQ_Old THEN
		IF MesDataIEC.IN_CmdQ = 0 THEN
			A1_PP.IN_CmdQ := 0;
		ELSIF MesDataIEC.IN_CmdQ < 2.802597E-45 THEN
			A1_PP.IN_CmdQ := 1;
		ELSIF MesDataIEC.IN_CmdQ < 3.9E-45 THEN
			A1_PP.IN_CmdQ := 2;
		ELSE
			A1_PP.IN_CmdQ := 3;
		END_IF
 
		CmdQ_Old 									:= MesDataIec.IN_CmdQ;
		bChange_CmdQ_Old							:= TRUE;
	ELSE                                    	
		bChange_CmdQ_Old							:= FALSE;
	END_IF
	
//	MesDataIEC.OUT_CmdQ 	:= A1_PP.IN_CmdQ;
	MesDataIEC.OUT_SetptPF	:= MesDataExd.OUT_SetptCosPhi;
	MesDataIEC.OUT_SetptU	:= MesDataExd.OUT_SetptU/1000;
	MesDataIEC.OUT_SetptQ	:= MesDataExd.MesData.OUT_SetptQ/1000;
END_METHOD

METHOD M_Execute
//////////////////
//  Method Calls 
/////////////////
VAR 
	// Method local variables (reinitialized at each cycle) 
	// EMULATOR

	
END_VAR
// READING AND WRITING CLOCK //

// PERMANENT CONDITIONS //
	M_CP() ; 
	
// METHODS CALLS //
	IF bInit THEN
		M_Init() ; 
		bInit:= FALSE ; 
	ELSIF CmdInit_G THEN 
		bInit:= TRUE ;
	END_IF

	M_IEC104(); 
	M_Evaluate() ; 
	
	////////////////////
	M_AlarmManagement();
END_METHOD

METHOD M_IEC104
//////////////////
//  Read Modbus Variable for PCS . 
/////////////////
VAR 
	// Method local variables (reinitialized at each cycle) 
	
	bTest: BOOL;
	KK: BYTE;
END_VAR
	
FB_IEC(
	IN_bEnable := TRUE , //Mesdata.MesCP_Read , 
	AODB := AODB , 
	memory := ADR(memory) , 
	IN_Local := MesDataIEC.OUT_MesLocal ) ;
END_METHOD

METHOD M_Init
VAR 

END_VAR

// Initialize autorization couplage to false
IF bBoot AND NOT A1_SUBMV.MesDataExd.MesData.MesState.1 THEN 
	MesDataExd.MesData.OUT_CmdAutCpl := FALSE ;  // A VOIR SI ON VEUT MEMORISER CET ETAT OU PAS AU DEMARRAGE. Le MesData est persistent.
	bBoot := FALSE ;
END_IF


///// INITIALIZE ////CstIPIEC104
// SERVER 1
	(* Configure protocol parameter *)
	FB_IEC.protPara.iK 				:= 12;(* default = 12 *)
	FB_IEC.protPara.iW 				:= 8;(* default = 8 *)
	FB_IEC.protPara.bThrottleMode 	:= TRUE;

	(* Configure system parameter *)
	FB_IEC.sysPara.asduAddr 		:= 1;
	FB_IEC.sysPara.bUsePCTime 		:= TRUE;
	FB_IEC.sysPara.bSyncTime 		:= TRUE;
	FB_IEC.sysPara.bSyncPCTime 		:= FALSE;
	FB_IEC.sysPara.bEndOfInit 		:= TRUE;
	FB_IEC.sysPara.bPerCyclic		:= TRUE;
	FB_IEC.sysPara.tPerCyclicBase	:= T#3S;
	FB_IEC.sysPara.bBackScan		:= TRUE;
	FB_IEC.sysPara.tBackScanCycle	:= T#3S;
	FB_IEC.sysPara.bPerFRZ			:= TRUE;
	FB_IEC.sysPara.tPerFRZCycle		:= T#15S;
	FB_IEC.sysPara.dbgMode 			:= (*IEC870_DEBUGMODE_ASDU OR*) IEC870_DEBUGMODE_DISABLED;

	(* Configure akuo iec104 parameter *)
	FB_IEC.akuoPara.iAOnb			:= 33 ; 
	FB_IEC.akuoPara.sLocalHost		:= CstIPIEC104 ; 
	

	(* Set point,  short floating point values *)
	initError := F_iecInitAOEntry( C_SE_NC_1, 1, 0, 0, MAP_AREA_MEMORY, 154, 0, AODB[32] );		//IN_SetptU 			AT%MB154  
	initError := F_iecInitAOEntry( C_SE_NC_1, 2, 0, 0, MAP_AREA_MEMORY, 158, 0, AODB[1] );		//IN_SetptP 			AT%MB158
	initError := F_iecInitAOEntry( C_SE_NC_1, 3, 0, 0, MAP_AREA_MEMORY, 162, 0, AODB[2] );		//IN_SetptQ 			AT%MB162
	initError := F_iecInitAOEntry( C_SE_NA_1, 4, 0, 0, MAP_AREA_MEMORY, 166, 0, AODB[3] );		//IN_CmdQ 				AT%MB166  
	initError := F_iecInitAOEntry( C_SE_NC_1, 5, 0, 0, MAP_AREA_MEMORY, 150, 0, AODB[0] );		//IN_CmdP1 				AT%MB150
	
	
		(* DP *)																												
//	initError := F_iecInitAOEntry( M_DP_TB_1, 100, IEC870_GRP_INROGEN, 0, MAP_AREA_MEMORY, 13, 0, AODB[] );			// 	OUT_MesPosCB_SubMV						      	
//	initError := F_iecInitAOEntry( M_DP_TB_1, 101, IEC870_GRP_INROGEN, 0, MAP_AREA_MEMORY, 13, 2, AODB[] );  		// 	OUT_MesPosSec_SubMV		       
//	initError := F_iecInitAOEntry( M_DP_TB_1, 102, IEC870_GRP_INROGEN, 0, MAP_AREA_MEMORY, 13, 4, AODB[] );  		//  OUT_MesPosEarth_SubMV	  

	initError := F_iecInitAOEntry( M_DP_TB_1, 103, IEC870_GRP_INROGEN OR IEC870_GRP_Background, 1 , MAP_AREA_MEMORY, 13, 6, AODB[ 4] );			// 	OUT_CmdPvF_On			  

	initError := F_iecInitAOEntry( M_DP_TB_1, 104, IEC870_GRP_INROGEN OR IEC870_GRP_background, 1 , MAP_AREA_MEMORY, 16, 2,  AODB[ 5] );	// 	OUT_CmdQvU	
	initError := F_iecInitAOEntry( M_DP_TB_1, 105, IEC870_GRP_INROGEN OR IEC870_GRP_Background, 1 , MAP_AREA_MEMORY, 14, 2,  AODB[ 6] );			// 	OUT_CmdPvF				  
	initError := F_iecInitAOEntry( M_DP_TB_1, 106, IEC870_GRP_INROGEN OR IEC870_GRP_Background, 1 , MAP_AREA_MEMORY, 14, 4,  AODB[ 7] );		// 	OUT_CmdQvU_On			  
	initError := F_iecInitAOEntry( M_DP_TB_1, 107, IEC870_GRP_INROGEN OR IEC870_GRP_Background, 1 , MAP_AREA_MEMORY, 14, 6,  AODB[ 8] );		// 	OUT_MesPosInter_33kV	  
	initError := F_iecInitAOEntry( M_DP_TB_1, 108, IEC870_GRP_INROGEN OR IEC870_GRP_Background, 1 , MAP_AREA_MEMORY, 15, 0,  AODB[ 9] );		// 	OUT_MesPosSecLinea_33kV	  
	initError := F_iecInitAOEntry( M_DP_TB_1, 109, IEC870_GRP_INROGEN OR IEC870_GRP_Background, 1 , MAP_AREA_MEMORY, 15, 2,  AODB[10] );		// 	OUT_MesPosSec_33kV		  
	initError := F_iecInitAOEntry( M_DP_TB_1, 110, IEC870_GRP_INROGEN OR IEC870_GRP_Background, 1 , MAP_AREA_MEMORY, 15, 4,  AODB[11] );		// 	OUT_MesPosGround_33kV	  
	initError := F_iecInitAOEntry( M_DP_TB_1, 111, IEC870_GRP_INROGEN OR IEC870_GRP_Background, 1 , MAP_AREA_MEMORY, 15, 6,  AODB[12] );		// 	OUT_MesPosInter_110kV	  
	initError := F_iecInitAOEntry( M_DP_TB_1, 112, IEC870_GRP_INROGEN OR IEC870_GRP_Background, 1 , MAP_AREA_MEMORY, 16, 0,  AODB[13] );		// 	OUT_MesPosSecLinea_110kV
                                               

(* Measured value , short floating point value *)	
	initError := F_iecInitAOEntry( M_ME_NC_1, 1000, IEC870_GRP_INROGEN OR IEC870_GRP_BACKGROUND, 1, MAP_AREA_MEMORY, 22	 , 0, AODB[14] );	//	OUT_MesP_33kV		 	AT%MB22	    
	initError := F_iecInitAOEntry( M_ME_NC_1, 1001, IEC870_GRP_INROGEN OR IEC870_GRP_Background, 1, MAP_AREA_MEMORY, 26	 , 0, AODB[15] );  //	OUT_MesQ_33kV			AT%MB26	     
	initError := F_iecInitAOEntry( M_ME_NC_1, 1002, IEC870_GRP_INROGEN OR IEC870_GRP_Background, 1, MAP_AREA_MEMORY, 30	 , 0, AODB[16] );  //	OUT_MesU12_33kV			AT%MB30	    
	initError := F_iecInitAOEntry( M_ME_NC_1, 1003, IEC870_GRP_INROGEN OR IEC870_GRP_Background, 1, MAP_AREA_MEMORY, 34	 , 0, AODB[17] );  //	OUT_MesI2_33kV 			AT%MB34	    
	initError := F_iecInitAOEntry( M_ME_NC_1, 1004, IEC870_GRP_INROGEN OR IEC870_GRP_Background, 1, MAP_AREA_MEMORY, 38	 , 0, AODB[18] );  //	OUT_MesP_110kV		 	AT%MB38	   
	initError := F_iecInitAOEntry( M_ME_NC_1, 1005, IEC870_GRP_INROGEN OR IEC870_GRP_Background, 1, MAP_AREA_MEMORY, 42	 , 0, AODB[19] );	//	OUT_MesQ_110kV			AT%MB42	    
	initError := F_iecInitAOEntry( M_ME_NC_1, 1006, IEC870_GRP_INROGEN OR IEC870_GRP_Background, 1, MAP_AREA_MEMORY, 46	 , 0, AODB[20] );  //	OUT_MesU12_110kV		AT%MB46	   
	initError := F_iecInitAOEntry( M_ME_NC_1, 1007, IEC870_GRP_INROGEN OR IEC870_GRP_Background, 1, MAP_AREA_MEMORY, 50	 , 0, AODB[21] );  //	OUT_MesI2_110kV 		AT%MB50	   
	initError := F_iecInitAOEntry( M_ME_NC_1, 1008, IEC870_GRP_INROGEN OR IEC870_GRP_Background, 1, MAP_AREA_MEMORY, 54	 , 0, AODB[22] );  //	OUT_SetptU				AT%MB54	       
	initError := F_iecInitAOEntry( M_ME_NC_1, 1009, IEC870_GRP_INROGEN OR IEC870_GRP_Background, 1, MAP_AREA_MEMORY, 58	 , 0, AODB[23] );	//	OUT_SetptPF				AT%MB58	      
	initError := F_iecInitAOEntry( M_ME_NC_1, 1010, IEC870_GRP_INROGEN OR IEC870_GRP_background, 1, MAP_AREA_MEMORY, 62	 , 0, AODB[24] );  //	OUT_SetptQ				AT%MB62	       
	initError := F_iecInitAOEntry( M_ME_NC_1, 1011, IEC870_GRP_INROGEN OR IEC870_GRP_background, 1, MAP_AREA_MEMORY, 66	 , 0, AODB[25] );  //	OUT_MesAvailability		AT%MB66	
	initError := F_iecInitAOEntry( M_ME_NC_1, 1012, IEC870_GRP_INROGEN OR IEC870_GRP_background, 1, MAP_AREA_MEMORY, 70	 , 0, AODB[26] );  //	OUT_MesPMax				AT%MB70	      
	initError := F_iecInitAOEntry( M_ME_NC_1, 1013, IEC870_GRP_INROGEN OR IEC870_GRP_background, 1, MAP_AREA_MEMORY, 74	 , 0, AODB[27] );  //	OUT_MesGTI				AT%MB74	       
	initError := F_iecInitAOEntry( M_ME_NC_1, 1014, IEC870_GRP_INROGEN OR IEC870_GRP_background, 1, MAP_AREA_MEMORY, 82	 , 0, AODB[28] );  //	OUT_MesTempPan			AT%MB82	    
	initError := F_iecInitAOEntry( M_ME_NC_1, 1015, IEC870_GRP_INROGEN OR IEC870_GRP_background, 1, MAP_AREA_MEMORY, 86	 , 0, AODB[29] );	//	OUT_MesGHI				AT%MB86	       
	initError := F_iecInitAOEntry( M_ME_NC_1, 1016, IEC870_GRP_INROGEN OR IEC870_GRP_background, 1, MAP_AREA_MEMORY, 90	 , 0, AODB[30] );  //	OUT_MesTempAmb			AT%MB90	    
//	initError := F_iecInitAOEntry( M_ME_NC_1, 1017, IEC870_GRP_background, 1, MAP_AREA_MEMORY, 94	 , 0, AODB[31] );  //	OUT_MesP_33kV_1			AT%MB94	   
//	initError := F_iecInitAOEntry( M_ME_NC_1, 1018, IEC870_GRP_background, 1, MAP_AREA_MEMORY, 98	 , 0, AODB[32] );  //	OUT_MesQ_33kV_1			AT%MB98	   
//	initError := F_iecInitAOEntry( M_ME_NC_1, 1019, IEC870_GRP_background, 1, MAP_AREA_MEMORY, 102    , 0, AODB[33] );	//	OUT_MesU_33kV_1			AT%MB102   
//	initError := F_iecInitAOEntry( M_ME_NC_1, 1020, IEC870_GRP_INROGEN OR IEC870_GRP_background, 1, MAP_AREA_MEMORY, 106    , 0, AODB[34] );  //	OUT_MesI_33kV_1			AT%MB106   
	initError := F_iecInitAOEntry( M_ME_NC_1, 1021, IEC870_GRP_INROGEN OR IEC870_GRP_background, 1, MAP_AREA_MEMORY, 110    , 0, AODB[31] );  //	OUT_MesTapPos			AT%MB110
END_METHOD

END_FUNCTION_BLOCK

// ---- 01_Equipement_Library/GRID/FB_GRID_MADI.TcPOU
FUNCTION_BLOCK FB_GRID_MADI EXTENDS FB_GRID_Base
//////////////////
// Grid Operator interface . Base FB
//////////////////
VAR_INPUT PERSISTENT
	// Parameters of the Object (instance specific) 

		ParamTONFiltering						: TIME:=T#500MS; 	(* Filtre tempo minimum avant validation de la commande (Filtrage du bruit)	*)
		ParamTONPulse							: TIME:=T#1S; 		(* Tempo to transform command to impulse .                                  *)
		{attribute 'OPC.UA.DA' := '1'}                                                                                                       
		ParamPmaxPark							: REAL;				(* Puissance max du park (Kw)                                               *)
		{attribute 'OPC.UA.DA' := '1'}                              
		ParamPminPark							: REAL ; 			(* puissance minimal du park                                                *)
		{attribute 'OPC.UA.DA' := '1'}                              
		ParamEmax								: REAL ; 			(* Maximal Contractual Energy .                                             *)
		                                                            
		ParamTempoComAlarm			: TIME 		:= T#10S;			(* Time before communication alarm	                                        *)
		
		
		
		MesDataExd				: GRID_MADI ; 
END_VAR


VAR_INPUT
	// I/O Inputs 
		//FROM AKSES
		IN_CmdAut_Cpl_other				: BOOL;
		IN_CmdDisconnect_other			: BOOL;	
		//IN_CmdConnect_other			: BOOL;	
		IN_CmdSoutirage_other			: BOOL;	
		IN_CmdInjection_other			: BOOL;			
		IN_CmdTest_other				: BOOL;	
		IN_CmdManualMode_other			: BOOL;
		IN_CmdManualModeOff_other		: BOOL;
	    IN_CmdToggleRead				: BOOL;	
		IN_ConnectAuthorizationLost		: BOOL; 

END_VAR 
VAR_OUTPUT
	//Child objects 17 OUtput
END_VAR



VAR
	//M_ALARMMANAGEMENT VARIABLES//                                                    								
		TON_ComAlarm							: TON;
		RS_ChargingAlarm						: RS;
	//M_EVALUATE VARIABLES//					
		//TON                       			
		TONConnectAuthorization					: TON;
		TONDisconnectOrder	        			: TON;
	    TONSoutirage	            			: TON;
	    TONTest	                				: TON;
	    TONModeManu				    			: TON;
		TONModeManuOff							: TON;
		TOF_ToS									: TOF;
                                                
                                                
		TONConnectAuthorizationPulse			: TON;
		TONDisconnectOrderPulse               	: TON;
	    TONModeManuPulse				        : TON;
		
		CheckCommand							: ARRAY[1..5] OF  FB_CheckCommand ;
		TON_CheckCommand						: ARRAY[1..5] OF TON ;
		
		OUT_MesEconnected						: REAL;// To be used for HMI only
		OUT_MesEmaxconnected					: REAL;
		OUT_MesIECServerFault					: BOOL;		
		
		RS_Soutirage_other						: RS;
		
	//M_Evaluate
		SetptP_old								: REAL;
		ParamPmax_old							: REAL ;
		ParamPmin_old							: REAL;		
                                        		
	// IEC 104                          		
	 	MesDataIEC								: IEC104_MADI;
		AODB 									: ARRAY[0..GVL_Cst.CstNbAOEntries] OF ST_IEC870_5_101AODBEntry ;
		memory 			AT%MB0					: ARRAY[0..79] OF BYTE;
		FB_IEC									: FB_IEC104ServerAkuo;(* Controlled station function block instance *)

	
	//M_INIT VARIABLES //
	//	bInit									: BOOL:= TRUE;	
		initError								: UDINT;
		bBoot									: BOOL := TRUE ; // Boolean that indicates a restart of the PLC .
	// M_EXECUTE VARIABLES //
        Trig_Cmd_Read							: R_TRIG;                                                                                        
		
		   		                    		
                     
				
END_VAR

METHOD M_AlarmManagement
//////////////////
// alarm and warning management
/////////////////

VAR 
	FB_AlarmCodeManager			: FB_AlarmCodeManager ; 
	

END_VAR
	TON_ComAlarm	(IN:= NOT( FB_IEC.eDTState =1 ) , PT:= ParamTempoComAlarm, 	Q=> MesDataExd.MesData.MesAlarmCom) ;	

	RS_ChargingAlarm(SET:= MesDataIEC.OUT_MesCharging , RESET1:= MesDataIEC.OUT_MesDischarging ) ; 
	
// ALARM CODE //
	FB_AlarmCodeManager(
		bAlarm1			:=MesDataIEC.IN_SetptP >MesDataIEC.IN_ParamPmax OR MesDataIEC.IN_SetptP < MesDataIEC.IN_ParamPmin, 	// Setpoint received outside of limits 
		bAlarm2			:=MesDataIEC.IN_Cmddouble.0 = MesDataIEC.IN_Cmddouble.1 , 												// Uncohetent not defined signal 
		bAlarm3			:=MesDataIEC.IN_Cmddouble.2 = MesDataIEC.IN_Cmddouble.3, 												// Uncoherent Start signal 
		bAlarm4			:=MesDataIEC.IN_Cmddouble.4 = MesDataIEC.IN_Cmddouble.5, 												// Uncoherent test signal
		bAlarm5			:=FALSE, 																								//
		bAlarm6			:=FALSE,                                                                                                //
		bAlarm7			:=FALSE,                                                                                                //
		bAlarm8			:=FALSE,                                                                                                //
		bAlarm9			:=FALSE, 																								//
		bAlarm10		:=FALSE,                                                                                                //
		bAlarm11		:=FALSE,                                                                                                //
		bAlarm12		:=FALSE,                                                                                                //
		bAlarm13		:=FALSE, 																								//
		bAlarm14		:=NOT MesDataExd.MesData.MesCP_Read,																				// IEC 104 Disabled.  
		bAlarm15		:= MesDataExd.MesData.MesAlarmCom, 						 															// Communication alarm with IEC 104 #COM
		wAlarmCode		=>MesDataExd.MesData.MesAlarmCode);

// WARNING CODE //
	FB_AlarmCodeManager(		
		bAlarm1			:=RS_ChargingAlarm.Q1 , 														//Monitoring direction : PP is charging
		bAlarm2			:=NOT RS_ChargingAlarm.Q1, 														//Monitoring direction : PP is discharging
		bAlarm3			:= MesDataIEC.OUT_MesEs, 														//Monitoring direction : Emergency stop     
		bAlarm4			:= MesDataIEC.OUT_MesLocal, 														//Monitoring direction : Local Mode
		bAlarm5			:= MesDataIEC.OUT_MesModeAuto_on, 												//Monitoring direction : Frequency regulation in progress
		bAlarm6			:= MesDataIEC.OUT_MesModeManuel_on, 												//Monitoring direction : Manual Mode is active
		bAlarm7			:= MesDataIEC.OUT_MesToS, 														//Monitoring direction : Techician on site
		bAlarm8			:= MesDataIEC.MesCentrale_Cpl, 													//Monitoring direction : PP is connected to the grid
		bAlarm9			:= MesDataIEC.MesCentrale_indispo, 												//Monitoring direction : PP is unavailable
		bAlarm10		:= MesDataIEC.MesSoutirage_on, 														//Monitoring direction : PP is started
		bAlarm11		:= MesDataIEC.OUT_MesIECServerFault, 											//Monitoring direction : IEC server fault   
		bAlarm12		:= MesDataIEC.OUT_MesFaultTeleCmd, 												//Monitoring direction : TC server fault
		bAlarm13		:= MesDataIEC.OUT_MesFaultTeleSgnl, 												//Monitoring direction : TS server fault             
		bAlarm14		:= MesDataIEC.OUT_MesFaultTeleMes, 												//Monitoring direction : TM server fault               
		bAlarm15		:= MesDataIEC.OUT_MesIncident       ,       										//Monitoring direction : Incident       
		wAlarmCode		=>MesDataExd.MesData.MesWarningCode);		

// EVENT CODE 1//

	FB_AlarmCodeManager(
		bAlarm1			:= MesDataIEC.IN_CmdAut_Cpl	, 					// Control direction : Coupling autorization request
		bAlarm2			:=FALSE	, 							            //
		bAlarm3			:= MesDataIEC.IN_CmdModeManuel	, 	            // Control direction : Manual Mode activation request 
		bAlarm4			:= MesDataIEC.IN_CmdDisconnect    , 	            // Control direction : PP disconnection request 
		bAlarm5			:= MesDataIEC.CmdSoutirage    , 	                    // Control direction : PP soutirage request  
		bAlarm6			:=FALSE, 	                                    //
		bAlarm7			:=FALSE, 	                                    //
		bAlarm8			:=FALSE, 	                                    //
		bAlarm9			:=FALSE   , 	                                //
		bAlarm10		:=FALSE, 	                                    //
		bAlarm11		:=FALSE, 	                                    //
		bAlarm12		:=FALSE   , 	                                //
		bAlarm13		:=FALSE   , 	                                //
		bAlarm14		:=FALSE, 	                                    //
		bAlarm15		:=FALSE, 	                                    //
		wAlarmCode		=>MesDataExd.MesData.MesEventCode);
END_METHOD

METHOD M_CP
VAR 

END_VAR


SUPER^.M_CP() ; 




Trig_Cmd_Read(CLK:=IN_CmdToggleRead);
	
IF Trig_Cmd_Read.Q THEN
	IN_CmdToggleRead := FALSE;
	MesDataExd.MesData.MesCP_Read := NOT MesDataExd.MesData.MesCP_Read;
END_IF
END_METHOD

METHOD M_Evaluate
//////////////////
//  Read Modbus Variable for PCS . 
/////////////////
VAR 
	// Method local variables (reinitialized at each cycle) 
	KK: INT;
	CalTos: BOOL;
	CalEs: BOOL;

	CalComEss: BOOL;



	

END_VAR
	// Update values to be sent through IEC 104 . 

	//MesDataIEC.MesStart_on := A1_PP.MesDataExd.MesData.MesState.2 ; 		// Ecrit par le protocole comme un acquittement
	//MesDataIEC.MesComTest_on := ; 								// ecrit par le protocole comme un acquittement .
	
MesDataIEC.MesCentrale_Cpl :=  A1_PP.MesData.MesState.2  ;									
MesDataIEC.MesCentrale_indispo := A1_PP.MesData.MesPP_Unavailable ; // Alarmes feu, arret urgence, mode local , UPS en decharge , Puissance dispo trop faible , 
MesDataIEC.MesDJOpen  :=  A1_SUBMV.A1_MainMVCB.MesDataExd.MesData.MesOpened; // DJ open
	
	
	
(*.MesDataIEC.OUT_MesDouble.0 := NOT MesDataIEC.MesStart_on ; 
.MesDataIEC.OUT_MesDouble.1 := MesDataIEC.MesStart_on ; *)
(*.MesDataIEC.OUT_MesDouble.2 := MesDataIEC.MesComTest_on ; 
.MesDataIEC.OUT_MesDouble.3 := NOT MesDataIEC.MesComTest_on ; *) 
MesDataIEC.OUT_MesDouble.4 := MesDataIEC.MesCentrale_Cpl ; 
MesDataIEC.OUT_MesDouble.5 := NOT MesDataIEC.MesCentrale_Cpl ;
MesDataIEC.OUT_MesDouble.6 := MesDataIEC.MesCentrale_indispo ; 
MesDataIEC.OUT_MesDouble.7 := NOT MesDataIEC.MesCentrale_indispo ;

MesDataIEC.OUT_MesDouble.0 := NOT MesDataIEC.MesDJOpen ; 
MesDataIEC.OUT_MesDouble.1 := MesDataIEC.MesDJOpen ; 	
	
	(*
	CalEs	:= FALSE ;
	CalTos	:= FALSE ;
	CalComEss := FALSE;
	
	FOR KK:= 1 TO CstNbEss DO 
		CalTos := CalTos OR AX_ESS[KK].A1_ToS.MesDataExd.MesData.MesAlarmState OR AX_ESS[KK].A1_DS_Bat.MesDataExd.MesData.MesAlarmState OR AX_ESS[KK].A1_Ds_Pcs.MesDataExd.MesData.MesAlarmState ;
		CalEs	:= CalEs OR AX_ESS[KK].A1_ES.MesDataExd.MesData.MesAlarmState ;
		CalComEss := CalComESS OR AX_ESS[KK].AX_Bat[1].MesDataExd.MesData.MesAlarmCom OR AX_ESS[KK].AX_Bat[1].MesDataExd.MesData.MesAlarmCom ;
	END_FOR
	
.MesDataIEC.OUT_MesLocal			:= A1_PP.ParamLocalMode ; 
.MesDataIEC.OUT_MesModeManuel_on := A1_PP.MesDataExd.MesData.CalManualMode  ;
.MesDataIEC.OUT_MesModeAuto_on	:= A1_PP.MesDataExd.MesData.CalFreqMode  ;
.MesDataIEC.OUT_MesCharging		:= A1_PP.MesDataExd.MesData.MesPbat < - A1_SUBMV.A1_PM_Aux.MesDataExd.MesData.MesP - 500 ;   // Charging more than the auxiliaries  ( keep some margin  ). 
.MesDataIEC.OUT_MesDischarging	:= A1_PP.MesDataExd.MesData.MesPbat > 500 ;
.MesDataIEC.OUT_MesEs			:= A1_SUBMV.A1_TOR_Es.MesDataExd.MesData.MesAlarmState OR CalEs ; 
	TOF_ToS(IN:= A1_SUBMV.A1_DS_LV.MesDataExd.MesData.MesAlarmState OR 	A1_SUBMV.A1_TOR_DsHT.MesDataExd.MesData.MesAlarmState OR CalTos , PT:= T#1H , Q =>MesDataIEC.OUT_MesToS	)  ; 	
.MesDataIEC.OUT_MesIncident		:=  (*A1_PP.MesDataExd.MesData.MesAlarmCode.0 OR*) A1_SUBMV.MesDataExd.MesData.MesAlarmCode.0 ; // Alarm on the PP or SUB_MV . 	
.MesDataIEC.OUT_MesFaultTeleMes	:= A1_SUBMV. AX_PM[1].MesDataExd.MesData.MesAlarmCom AND A1_SUBMV.AX_PM[2].MesDataExd.MesData.MesAlarmCom OR CalComEss; // Si defaut de com sur un des signaux de la telemesure . 	
.MesDataIEC.OUT_MesFaultTeleCmd	:= CheckCommand[1].bWarning OR CheckCommand[2].bWarning OR CheckCommand[3].bWarning OR CheckCommand[4].bWarning OR CheckCommand[5].bWarning  ; // Si defaut d	
	/.MesDataIEC.OUT_MesFaultTeleSgnl	:=   ; // Si defaut d ecriture modbus des setpoint de P . 
	OUT_MesIECServerFault				:= SEL(CstPLCBackup ,NOT MAIN.OUT_CalRunningPLC_IO  ,MAIN.OUT_CalRunningPLC_IO ) ; // NOT MesDataExd.MesData.MesCP_Read  ; // Define nwhich PA is active ( False  = PA 1  , else PA 2 )  
.MesDataIEC.OUT_MesIECServerFault	:= OUT_MesIECServerFault ;


	OUT_MesEconnected					:= A1_PP.MesDataExd.MesData.OUT_Econnected / 1000 ;	
.MesDataIEC.OUT_MesEconnected 		:= OUT_MesEconnected ;
	OUT_MesEmaxconnected 				:= A1_PP.MesDataExd.MesData.OUT_Enomconnected / 1000 ;			// MWh . Capacité maximale connectée ( taking account 12MWh max , and soc security .  
.MesDataIEC.OUT_MesEmaxconnected 	:= OUT_MesEmaxconnected; 
	
.MesDataIEC.OUT_MesP 			:= 	 A1_PP.MesDataExd.MesData.MesPbat /1000 ;		// MW
.MesDataIEC.OUT_MesQ 			:= 	 A1_PP.MesDataExd.MesData.MesQbat/1000 ;	// MVAr
.MesDataIEC.OUT_MesU_HTA 		:=	 A1_PP.MesDataExd.MesData.MesU/1000;		// kV
.MesDataIEC.OUT_MesFreq 			:= 	 A1_SUBMV.MesDataExd.MesData.MesFreq;		// Hz
.MesDataIEC.OUT_MesPdispo_inj 	:=  A1_PP.MesDataExd.MesData.OUT_SetptPmax  /1000 ; // MW
.MesDataIEC.OUT_MesPdispo_abs 	:=   A1_PP.MesDataExd.MesData.OUT_SetptPmin /1000 ; // MW 
*)
	// TREAT COMMANDS 
	// FAIRE DES IMPULSIONS SUR LES COMMANDES . 

	// Double point commands. 
MesDataIEC.CmdSoutirage := MesDataIEC.IN_Cmddouble.3 ;
MesDataIEC.CmdTest := MesDataIEC.IN_Cmddouble.4 ; 
	
	//Filtering Input
		TONConnectAuthorization	(IN:= MesDataIEC.IN_CmdAut_Cpl,PT:=ParamTONFiltering);
		TONDisconnectOrder		(IN:= MesDataIEC.IN_CmdDisconnect,PT:=ParamTONFiltering);		
		TONSoutirage	(IN:= MesDataIEC.CmdSoutirage,PT:=ParamTONFiltering);	
		TONTest	(IN:= MesDataIEC.CmdTest,PT:=ParamTONFiltering);	
		TONModeManu			(IN:= MesDataIEC.IN_CmdModeManuel,PT:=ParamTONFiltering);
		TONModeManuOff			(IN:= MesDataIEC.IN_CmdModeManuelOff,PT:=ParamTONFiltering);			



	// Impulsions
		TONConnectAuthorizationPulse	(IN:=TONConnectAuthorization.Q,PT:=ParamTONPulse);
		TONDisconnectOrderPulse		(IN:=TONDisconnectOrder.Q	,PT:=ParamTONPulse);		
		TONModeManuPulse		(IN:=TONModeManu.Q,PT:=ParamTONPulse);	

	RS_Soutirage_other(SET:=IN_CmdSoutirage_other , RESET1:=IN_CmdInjection_other (*OR MesDataExd.MesData.OUT_CmdDisconnect*)) ; 
	
	(*Autorisation de couplage*)
	IF TONConnectAuthorization.Q AND NOT A1_PP.ParamLocalMode OR A1_PP.ParamLocalMode AND IN_CmdAut_Cpl_other THEN
	MesDataExd.MesData.OUT_CmdAutCpl := TRUE ;
	MesDataExd.MesData.OUT_CmdDisconnect := FALSE ; 
		IF TONConnectAuthorizationPulse.Q THEN 
		MesDataIEC.IN_CmdAut_Cpl := FALSE ; // Reinitialize to false the input to get an impulse. 
		END_IF
	END_IF
	IF IN_ConnectAuthorizationLost THEN  //IN_Long_GTE_Fault OR IN_C13_100_Fault OR IN_UnknownFault OR IN_3GTE_Fault  OR CmdDecouplage 
	MesDataExd.MesData.OUT_CmdAutCpl := FALSE ;
	END_IF
	
	IF TONDisconnectOrder.Q AND NOT A1_PP.ParamLocalMode OR A1_PP.ParamLocalMode AND IN_CmdDisconnect_other THEN 
	MesDataExd.MesData.OUT_CmdDisconnect := TRUE ; 
	MesDataExd.MesData.OUT_CmdAutCpl := FALSE ;
		IF TONDisconnectOrderPulse.Q THEN 
		MesDataIEC.IN_CmdDisconnect := FALSE ; // Reinitialize to false the input to get an impulse.
		END_IF
	END_IF
	//  MesDataExd.MesData.OUT_CmdAut_Cpl := TONConnectAuthorization.Q OR A1_PP.ParamLocalMode AND IN_CmdAut_Cpl_other ; 	// Impulse // ADD LOCAL ONLY 

	IF 	TONModeManuPulse.Q 	AND NOT A1_PP.ParamLocalMode THEN 
	MesDataIEC.IN_CmdModeManuel := FALSE ; // Reinitialize to false the input to get an impulse.
	END_IF
	
	//  MesDataExd.MesData.OUT_CmdDisconnect := TONDisconnectOrder.Q 	OR A1_PP.ParamLocalMode AND IN_CmdDisconnect_other		; 
(*
MesDataExd.MesData.OUT_CmdModeManuel := TONModeManu.Q 	AND NOT A1_PP.ParamLocalMode		OR A1_PP.ParamLocalMode AND IN_CmdManualMode_other	; 	// Impulse
MesDataExd.MesData.OUT_CmdModeManuelOff := TONModeManuOff.Q 	AND NOT A1_PP.ParamLocalMode		OR A1_PP.ParamLocalMode AND IN_CmdManualModeOff_other	; 	// Impulse
MesDataExd.MesData.OUT_CmdSoutirage := (TONSoutirage.Q 		AND NOT A1_PP.ParamLocalMode 		OR  A1_PP.ParamLocalMode AND	RS_Soutirage_other.Q1) AND NOT MesDataExd.MesData.OUT_CmdDisconnect ;	// True / False . 
MesDataExd.MesData.OUT_CmdTest := TONTest.Q 		AND NOT A1_PP.ParamLocalMode			OR A1_PP.ParamLocalMode AND IN_CmdTest_other		; 
	*)
	// Write value only on change . 
	IF MesDataIEC.IN_SetptP <> SetptP_old THEN 
	MesDataExd.MesData.OUT_SetptP 				:= MesDataIEC.IN_SetptP *1000  ;  
		SetptP_old := MesDataIEC.IN_SetptP ; 
	END_IF

(*	IF MesDataIEC.IN_ParamPmax <> ParamPmax_old THEN 
	MesDataExd.MesData.OUT_ParamPmax			:=	MIN(MesDataIEC.IN_ParamPmax*1000 , ParamPmaxPark)  ;  
		ParamPmax_old := MesDataIEC.IN_ParamPmax   ; 
	END_IF	
	IF MesDataIEC.IN_ParamPmin <> ParamPmin_old THEN 
	MesDataExd.MesData.OUT_ParamPmin				:=	MAX( MesDataIEC.IN_ParamPmin*1000, ParamPminPark)   ;  
		ParamPmin_old := MesDataIEC.IN_ParamPmin ; 
	END_IF	
*)

	// Detect if command is not applied  
	// Start 
	TON_CheckCommand[1](IN:= CheckCommand[1].bWarning , PT:= T#2S ) ; 
	CheckCommand[1](
		bCmd		:= MesDataExd.MesData.OUT_CmdAutCpl  ,
		bMes		:= A1_PP.MesData.MesState.2 , 		// Compare with the modbus feedback on equipement . 
		bReset		:= TON_CheckCommand[1].Q,		// Reset after 2 se
		bImpulsion	:= TRUE , 
		T			:= T#120S ) ;
(*		
	// Stop Mode 
	TON_CheckCommand[2](IN:= CheckCommand[2].bWarning , PT:= T#2S ) ; 
	CheckCommand[2](
		bCmd		:=  NOT MesDataExd.MesData.OUT_CmdSoutirage ,
		bMes		:= A1_PP.MesDataExd.MesData.MesState.0 , 		// Compare with the modbus feedback on equipement . 
		bReset		:=TON_CheckCommand[2].Q ,
		bImpulsion	:= TRUE , 
		T			:= T#5S ) ;	
	*)
	// Disconnect 
	TON_CheckCommand[3](IN:= CheckCommand[3].bWarning , PT:= T#2S ) ; 
	CheckCommand[3](
		bCmd		:= MesDataExd.MesData.OUT_CmdDisconnect,
		bMes		:= A1_PP.MesData.MesState.0 , 		// Compare with the modbus feedback on equipement . 
		bReset		:= TON_CheckCommand[3].Q,
		bImpulsion	:= TRUE , 
		T			:= T#5S ) ;	
	
	// Autorization couplage 
	TON_CheckCommand[4](IN:= CheckCommand[4].bWarning , PT:= T#2S ) ; 
	CheckCommand[4](
		bCmd		:= MesDataExd.MesData.OUT_CmdAutCpl ,
		bMes		:= A1_SUBMV.MesDataExd.MesData.MesClosed_ALOFeederMVCB AND A1_SUBMV.MesDataExd.MesData.MesClosed_ALOFeederMVCB , 		// Compare with the modbus feedback on equipement . 
		bReset		:= TON_CheckCommand[4].Q,
		bImpulsion	:= TRUE , 
		T			:= T#5S ) ;
		
		(*
	// Manual Mode 
	TON_CheckCommand[5](IN:= CheckCommand[5].bWarning , PT:= T#2S ) ; 
	CheckCommand[5](
		bCmd		:= MesDataExd.MesData.OUT_CmdModeManuel ,
		bMes		:= A1_PP.MesDataExd.MesData.CalManualMode , 		// Compare with the modbus feedback on equipement . 
		bReset		:=TON_CheckCommand[5].Q ,
		bImpulsion	:= TRUE , 
		T			:= T#1S ) ;	
		
		*)
END_METHOD

METHOD M_Execute
//////////////////
//  Method Calls 
/////////////////
VAR 
	// Method local variables (reinitialized at each cycle) 
	// EMULATOR

	
END_VAR
// READING AND WRITING CLOCK //

// PERMANENT CONDITIONS //
	M_CP() ; 
	
// METHODS CALLS //
	IF bInit THEN
		M_Init() ; 
		bInit:= FALSE ; 
	ELSIF CmdInit_G THEN 
		bInit:= TRUE ;
	END_IF

	M_IEC104(); 
	M_Evaluate() ; 
	
	////////////////////
	M_AlarmManagement();
END_METHOD

METHOD M_IEC104
//////////////////
//  Read Modbus Variable for PCS . 
/////////////////
VAR 
	// Method local variables (reinitialized at each cycle) 
	
	bTest: BOOL;
	KK: BYTE;
END_VAR
	
FB_IEC(
	IN_bEnable := TRUE , //MesCP_Read , 
	AODB := AODB , 
	memory := ADR(memory) , 
	IN_Local := MesDataIEC.OUT_MesLocal ) ;
END_METHOD

METHOD M_Init
VAR 


END_VAR

// Initialize autorization couplage to false
IF bBoot AND NOT A1_SUBMV.MesDataExd.MesData.MesState.1 THEN 
	MesDataExd.MesData.OUT_CmdAutCpl := FALSE ;  // A VOIR SI ON VEUT MEMORISER CET ETAT OU PAS AU DEMARRAGE. Le.MesDataExd.MesData.est persistent.
	bBoot := FALSE ;
END_IF


///// INITIALIZE ////CstIPIEC104
// SERVER 1
	(* Configure protocol parameter *)
	FB_IEC.protPara.iK 				:= 12;(* default = 12 *)
	FB_IEC.protPara.iW 				:= 8;(* default = 8 *)
	FB_IEC.protPara.bThrottleMode 	:= TRUE;

	(* Configure system parameter *)
	FB_IEC.sysPara.asduAddr 		:= 1;
	FB_IEC.sysPara.bUsePCTime 		:= TRUE;
	FB_IEC.sysPara.bSyncTime 		:= TRUE;
	FB_IEC.sysPara.bSyncPCTime 		:= FALSE;
	FB_IEC.sysPara.bEndOfInit 		:= TRUE;
	FB_IEC.sysPara.bPerCyclic		:= TRUE;
	FB_IEC.sysPara.tPerCyclicBase	:= T#3S;
	FB_IEC.sysPara.bBackScan		:= FALSE;
	FB_IEC.sysPara.tBackScanCycle	:= T#3S;
	FB_IEC.sysPara.bPerFRZ			:= TRUE;
	FB_IEC.sysPara.tPerFRZCycle		:= T#15S;
	FB_IEC.sysPara.dbgMode 			:= (*IEC870_DEBUGMODE_ASDU OR*) IEC870_DEBUGMODE_DEVSTATE;

	(* Configure akuo iec104 parameter *)
	FB_IEC.akuoPara.iAOnb			:= 33 ; 
	FB_IEC.akuoPara.sLocalHost		:= CstIPIEC104 ; 
	
	initError := F_iecInitAOEntry( M_SP_TB_1, 12, IEC870_GRP_INROGEN, 0,  MAP_AREA_MEMORY, 10, 0, AODB[0] );		//OUT_MesLocal		       
	initError := F_iecInitAOEntry( M_SP_TB_1, 13, IEC870_GRP_INROGEN, 0,  MAP_AREA_MEMORY, 10, 1, AODB[1] );		//OUT_MesModeManuel_on
	initError := F_iecInitAOEntry( M_SP_TB_1, 14, IEC870_GRP_INROGEN, 0,  MAP_AREA_MEMORY, 10, 2, AODB[2] );      //OUT_MesModeAuto_on	 
	initError := F_iecInitAOEntry( M_SP_TB_1, 15, IEC870_GRP_INROGEN, 0,  MAP_AREA_MEMORY, 10, 3, AODB[3] );	    //OUT_MesCharging		   
	initError := F_iecInitAOEntry( M_SP_TB_1, 16, IEC870_GRP_INROGEN, 0,  MAP_AREA_MEMORY, 10, 4, AODB[4] );	    //OUT_MesDischarging	 
	initError := F_iecInitAOEntry( M_SP_TB_1, 20, IEC870_GRP_INROGEN, 0,  MAP_AREA_MEMORY, 10, 5, AODB[5] );      //OUT_MesEs			        
	initError := F_iecInitAOEntry( M_SP_TB_1, 21, IEC870_GRP_INROGEN, 0,  MAP_AREA_MEMORY, 10, 6, AODB[6] );	    //OUT_MesToS			       
	initError := F_iecInitAOEntry( M_SP_TB_1, 19, IEC870_GRP_INROGEN, 0,  MAP_AREA_MEMORY, 10, 7, AODB[7] );	    //OUT_MesIncident			   
	initError := F_iecInitAOEntry( M_SP_TB_1, 37, IEC870_GRP_INROGEN, 0,  MAP_AREA_MEMORY, 11, 0, AODB[8] );	    //OUT_MesFaultTeleMes		
	initError := F_iecInitAOEntry( M_SP_TB_1, 38, IEC870_GRP_INROGEN, 0,  MAP_AREA_MEMORY, 11, 1, AODB[9] );	    //OUT_MesFaultTeleCmd		
	initError := F_iecInitAOEntry( M_SP_TB_1, 39, IEC870_GRP_INROGEN, 0,  MAP_AREA_MEMORY, 11, 2, AODB[10] );	    //OUT_MesFaultTeleSgnl	
	initError := F_iecInitAOEntry( M_SP_TB_1, 41, IEC870_GRP_INROGEN, 0,  MAP_AREA_MEMORY, 11, 3, AODB[11] );	    //OUT_MesIECServerFault

		(* TSD *)
	initError := F_iecInitAOEntry( M_DP_TB_1, 43, IEC870_GRP_INROGEN, 0, MAP_AREA_MEMORY, 61, 2, AODB[12] );	//MesSoutirage_on			      	
	initError := F_iecInitAOEntry( M_DP_TB_1, 44, IEC870_GRP_INROGEN, 0, MAP_AREA_MEMORY, 61, 4, AODB[13] );   //MesComTest_on		     
	initError := F_iecInitAOEntry( M_DP_TB_1, 17, IEC870_GRP_INROGEN, 0, MAP_AREA_MEMORY, 12, 4, AODB[14] );   //MesCentrale_Cpl		   
	initError := F_iecInitAOEntry( M_DP_TB_1, 22, IEC870_GRP_INROGEN, 0, MAP_AREA_MEMORY, 12, 6, AODB[15] );	//MesCentrale_indispo	
	initError := F_iecInitAOEntry( M_DP_TB_1, 51, IEC870_GRP_INROGEN, 0, MAP_AREA_MEMORY, 12, 0, AODB[33] );   //MesDJOpen		   


	
	(* Measured value , short floating point value *)
	initError := F_iecInitAOEntry( M_ME_NC_1, 5, IEC870_GRP_INROGEN OR IEC870_GRP_PERCYC , 1, MAP_AREA_MEMORY, 42, 0, AODB[16] );	// OUT_MesSoC 			    
	initError := F_iecInitAOEntry( M_ME_NC_1, 6, IEC870_GRP_INROGEN OR IEC870_GRP_PERCYC , 1, MAP_AREA_MEMORY, 14, 0, AODB[17] );  // OUT_MesSoH 			    
	initError := F_iecInitAOEntry( M_ME_NC_1, 1, IEC870_GRP_INROGEN OR IEC870_GRP_PERCYC , 1, MAP_AREA_MEMORY, 18, 0, AODB[18] );  // OUT_MesP 			      
	initError := F_iecInitAOEntry( M_ME_NC_1, 2, IEC870_GRP_INROGEN OR IEC870_GRP_PERCYC , 1, MAP_AREA_MEMORY, 22, 0, AODB[19] );  // OUT_MesQ 			      
	initError := F_iecInitAOEntry( M_ME_NC_1, 3, IEC870_GRP_INROGEN OR IEC870_GRP_PERCYC , 1, MAP_AREA_MEMORY, 26, 0, AODB[20] );  // OUT_MesU_HTA 		   
	initError := F_iecInitAOEntry( M_ME_NC_1, 4, IEC870_GRP_INROGEN OR IEC870_GRP_PERCYC , 1, MAP_AREA_MEMORY, 30, 0, AODB[21] );	// OUT_MesFreq 		    
	initError := F_iecInitAOEntry( M_ME_NC_1, 7, IEC870_GRP_INROGEN OR IEC870_GRP_PERCYC , 1, MAP_AREA_MEMORY, 34, 0, AODB[22] );  // OUT_MesPdispo_inj 
	initError := F_iecInitAOEntry( M_ME_NC_1, 8, IEC870_GRP_INROGEN OR IEC870_GRP_PERCYC , 1, MAP_AREA_MEMORY, 38, 0, AODB[23] );  // OUT_MesPdispo_abs 

	(* Single commands *)
	initError := F_iecInitAOEntry( C_SC_TA_1, 30, 0, 0, MAP_AREA_MEMORY, 60, 0, AODB[24] );	//	IN_CmdModeManuel
	initError := F_iecInitAOEntry( C_SC_TA_1, 31, 0, 0, MAP_AREA_MEMORY, 60, 1, AODB[27] );	//	IN_CmdModeManuelOff
	initError := F_iecInitAOEntry( C_SC_TA_1, 32, 0, 0, MAP_AREA_MEMORY, 60, 2, AODB[25] );   //  IN_CmdAut_Cpl	  
	initError := F_iecInitAOEntry( C_SC_TA_1, 33, 0, 0, MAP_AREA_MEMORY, 60, 3, AODB[26] );	//	CmdDisconnect	
	
	(* Double commands *)
	initError := F_iecInitAOEntry( C_DC_TA_1, 26, 0, 0, MAP_AREA_MEMORY, 61, 2, AODB[28] );	//  CmdSoutirage		    
	initError := F_iecInitAOEntry( C_DC_TA_1, 27, 0, 0, MAP_AREA_MEMORY, 61, 4, AODB[29] );	//  CmdTest			    

	(* Set point,  short floating point values *)
	initError := F_iecInitAOEntry( C_SE_TC_1, 36, 0, 0, MAP_AREA_MEMORY, 72, 0, AODB[30] );		//IN_SetptP 		 
	initError := F_iecInitAOEntry( C_SE_TC_1, 34, 0, 0, MAP_AREA_MEMORY, 64, 0, AODB[31] );		//IN_ParamPmax 
	initError := F_iecInitAOEntry( C_SE_TC_1, 35, 0, 0, MAP_AREA_MEMORY, 68, 0, AODB[32] );		//IN_ParamPmin
END_METHOD

END_FUNCTION_BLOCK

// ---- 01_Equipement_Library/Fan/FB_Fan_Basic.TcPOU
FUNCTION_BLOCK FB_Fan_Basic
// Function Block to ensure fan control 

VAR_INPUT PERSISTENT
	ParamNbSensors			: INT;				(* Number of temperature sensors*)
	{attribute 'OPC.UA.DA' := '1'} 
	ParamTemphigh 			: REAL := 35;		(*  (C)High temperature to trigger the fan*)
	{attribute 'OPC.UA.DA' := '1'} 
	ParamTemplow 			: REAL := 30;		(*  (C)Low temperature to trigger the fan*)
END_VAR
	
VAR_INPUT           	
	IN_LocalHour 	    	: TIMESTRUCT;	// 
	IN_ForceRun				: BOOL;			//
	IN_ForceStop			: BOOL; 		//
	IN_Tmp1_IO 				: REAL; 	    //  Temperature sensor 1
	IN_Tmp2_IO				: REAL;	    	//  Temperature sensor 2

	// Commands and setpoints 
	IN_CmdReset_L			: BOOL;			// (NA) External Reset Command
	
	MesDataExd				: Fan_Standard;	
END_VAR             	
VAR_OUTPUT          	
	OUT_Run_IO				: BOOL;
END_VAR             	
VAR                 	
	bInit					: BOOL := TRUE;		 // Booleen d'initialisation
	bTmp1_OK				: BOOL;				 // Booléen de test si les valeurs remontées par les capteurs de températures remontent une donnée correcte
	bTmp2_OK				: BOOL;
	bTmp_OK 				: BOOL;
	fTmp_PT					: REAL;

	// State Mananger //
	MesState				: BYTE;  // Cal 
	
END_VAR

VAR PERSISTENT
	MesStartTime 			: WORD := 9;
	MesStopTime				: WORD := 19;
END_VAR

METHOD M_AlarmManagement
//////////////////
// Generates object alarms and manages resets. 
//////////////////

VAR 
	// Method local variables (reinitialized at each cycle) 
	FB_AlarmCodeManager		: FB_AlarmCodeManager ;  
END_VAR

	IF ParamNbSensors = 1 THEN
		IN_Tmp2_IO := IN_Tmp2_IO;
	END_IF
	bTmp1_OK 	:= IN_Tmp1_IO < 70 AND IN_Tmp1_IO > -10;
	bTmp2_OK 	:= IN_Tmp2_IO < 70 AND IN_Tmp2_IO > -10;
	bTmp_OK 	:=  bTmp1_OK OR bTmp2_OK;
	IF bTmp1_OK AND bTmp2_OK THEN
		fTmp_PT 	:= (IN_Tmp1_IO +  IN_Tmp2_IO )/2;
	ELSE
		fTmp_PT 	:= (IN_Tmp1_IO * BOOL_TO_BYTE(bTmp1_OK) + IN_Tmp2_IO * BOOL_TO_BYTE(bTmp2_OK));
	END_IF
	// Déclenchement du ventilateur
	// Boucle de sécurité sur les heures de fonctionnement
	IF IN_LocalHour.wHour > MesStartTime AND IN_LocalHour.wHour <MesStopTime AND bTmp_OK  THEN
		IF fTmp_PT > ParamTemphigh  THEN
			OUT_Run_IO := TRUE;
		END_IF
		
		IF fTmp_PT < ParamTemplow THEN
			OUT_Run_IO := FALSE;
		END_IF
		
	END_IF
	OUT_Run_IO := (OUT_Run_IO OR IN_ForceRun) AND NOT IN_ForceStop;
	
// ALARM CODE //
	FB_AlarmCodeManager(
		bAlarm1				:= IN_ForceStop,		//		Fans are forced to Stop
		bAlarm2				:= FALSE,//
		bAlarm3				:= FALSE,//
		bAlarm4				:= FALSE,//
		bAlarm5				:= FALSE,//
		bAlarm6				:= FALSE,//
		bAlarm7				:= FALSE,//
		bAlarm8				:= FALSE,//
		bAlarm9				:= FALSE,//
		bAlarm10			:= FALSE,//
		bAlarm11			:= FALSE,//
		bAlarm12			:= FALSE,//		
		bAlarm13			:= FALSE,//				
		bAlarm14			:= FALSE,//			
		bAlarm15			:= FALSE,//
		wAlarmCode			=>MesDataExd.MesData.MesAlarmCode);
			
// WARNING CODE //
	FB_AlarmCodeManager(
		bAlarm1				:= NOT bTmp_OK, // Temperature sensors are not working
		bAlarm2				:= FALSE,//
		bAlarm3				:= FALSE,//
		bAlarm4				:= FALSE,//
		bAlarm5				:= FALSE,//
		bAlarm6				:= FALSE,//
		bAlarm7				:= FALSE,//
		bAlarm8				:= FALSE,//
		bAlarm9				:= FALSE,//
		bAlarm10			:= FALSE,//
		bAlarm11			:= FALSE,//
		bAlarm12			:= FALSE,//
		bAlarm13			:= FALSE,//
		bAlarm14			:= FALSE,//
		bAlarm15			:= FALSE,//
		wAlarmCode			=>MesDataExd.MesData.MesWarningCode);
		
// EVENT CODE //

	FB_AlarmCodeManager(
		bAlarm1			:= OUT_Run_IO,  // Fans are requested to run
		bAlarm2			:= IN_ForceRun, // Fans are forced to run
		bAlarm3			:= FALSE,//
		bAlarm4			:= FALSE,//
		bAlarm5			:= FALSE,//
		bAlarm6			:= FALSE,//
		bAlarm7			:= FALSE,//
		bAlarm8			:= FALSE,//
		bAlarm9			:= FALSE,//
		bAlarm10		:= FALSE,//
		bAlarm11		:= FALSE,//
		bAlarm12		:= FALSE,//
		bAlarm13		:= FALSE,//
		bAlarm14		:= FALSE,//
		bAlarm15		:= FALSE,//
		wAlarmCode		=>MesDataExd.MesData.MesEventCode);
END_METHOD

METHOD M_Evaluate
//////////////////
// Evaluate available Powers and AMG characteristics . 
/////////////////

VAR 
	
END_VAR
MesDataExd.MesData.MesModeRun		:=	OUT_Run_IO;
MesDataExd.MesData.MesTemp 			:= 	fTmp_PT ; 
MesDataExd.Mesdata.MesStartTime 	:=	MesStartTime ;
MesDataExd.Mesdata.MesStopTime 		:=	MesStopTime ;
END_METHOD

METHOD M_Execute : BOOL
VAR_INPUT
END_VAR
IF NOT bInit THEN
	M_Init();

ELSIF CmdInit_G  OR IN_CmdReset_L THEN
	bInit := TRUE;
END_IF


M_StateManager();
M_Evaluate();
END_METHOD

METHOD M_Init : BOOL
VAR_INPUT
END_VAR



// Boucle d'initalisation des variables de température pour séléctionner une valeur de température
	OUT_Run_IO := FALSE;

	
	bInit := FALSE;
END_METHOD

METHOD M_StateManager
//////////////////
// Detect which is the state of the inverter. IF loss of communication MesState =0 , the last inverter state is kept .  
/////////////////

VAR 
	// Method local variables (reinitialized at each cycle) 

	
END_VAR
// OPERATIONNAL INDEX //
IF OUT_Run_IO THEN 
	MesState.2 := 1;
ELSE
	MesState.0 := 1;
END_IF
END_METHOD

END_FUNCTION_BLOCK

// ---- 01_Equipement_Library/HVAC/FB_HVAC_MeAcMbs1.TcPOU
FUNCTION_BLOCK FB_HVAC_MeAcMbs1 EXTENDS FB_HVAC_Base
VAR_INPUT PERSISTENT
	ParamTempoComAlarm						: TIME 		:= T#10S ; 	(* (s) Config : Tempo to detect LOC Alarm	*)
	{attribute 'OPC.UA.DA' := '1'}                                  
	ParamUnitID								: BYTE  	:= 1 ; 		(* (NA) Modbus Unit ID                           *)
	ParamPriority							: UINT;					(* (NA) Level of priority in the HVAC pool       *)
	
	ParamTimeOut							: TIME 		:= T#3S;	(* (NA) Modbus Timeout                           *)
	
	ParamTempMin							: REAL := 16; 		(* (°C) Minimal temperature setpoint allowed by device *)
	ParamTempMax							: REAL := 32; 		(* (°C) Maximal temperature setpoint allowed by device *)
	ParamNumEss								: UINT;				(* (NA) Number of the corresponding ESS *)
	
END_VAR

VAR_INPUT	
	IN_SetptTemp							: REAL:=22;
	IN_SetptHygro							: REAL;
	IN_CmdStart								: BOOL;
	IN_CmdStop								: BOOL;
	IN_CmdReset								: BOOL;

	IN_CmdReleaseStop_OPC					: BOOL ; // Manual Cmd. Non prioritaire sur le mode auto. 
	IN_CmdStop_OPC							: BOOL ; // Manual Cmd .Prioriatire sur le mode auto . Dévérouillage seulement sur ordre de start manual.  
	
			MesDataExd						: HVAC_MeAcMbs1;
END_VAR

VAR
	
	//M_ALARMMANAGEMENT VARIABLES 
		TON_ComAlarm				: TON ; 												// Tempo before detecting loss of communication. 
	


		
	//M_READ VARIABLES//
		bReadError						: BOOL;
		bReadCompleted 					: BOOL;
		bReadBusy						: BOOL;
		InputStructRead 				: Struct_InputRTU;
		TRIG_Read						: R_TRIG;
		TRIG_Write						: R_TRIG;
		
		
		bWriteError						: ARRAY[1..2] OF BOOL;
		bWriteCompleted 				: ARRAY[1..2] OF BOOL;
		bWriteBusy						: ARRAY[1..2] OF BOOL;
		InputStructWrite 				: ARRAY[1..2] OF Struct_InputRTU;
		                            	
		MesBlock1_Temp 					: ARRAY[1..125]  OF WORD; 		// (NA) Temporary Block with multiple modbus reading (Caution : Double Word variables)
		

		WordToWrite1					: WORD;
		WordToWrite2					: WORD;
		WordToWrite1_Old				: WORD;
		WordToWrite2_Old				: WORD;
	                                 
	
		RS_StartStop					: RS ; 
	
		R_TrigState						: R_TRIG;
		F_TrigState						: F_TRIG;
		TimeStart						: TIME;
		TimeNotStart					: TIME;
		
END_VAR
VAR_OUTPUT PERSISTENT
	          			
END_VAR

METHOD M_AlarmManagement : BOOL
VAR_INPUT
END_VAR

VAR
	FB_AlarmCodeManager			: FB_AlarmCodeManager ;
	CMWarning: BOOL;
	CMAlarm: BOOL;
	MesWarningCom: BOOL;
	WriteAlarm: BOOL;
END_VAR
		CMWarning 		:= bWriteError[1] OR bWriteError[2] OR bReadError;
		CMAlarm			:= bWriteError[1] AND bWriteError[2] AND bReadError;
		
	// Warning
	MesWarningCom 		:= CMWarning ; 											//
	//Alarm
	TON_ComAlarm(IN:= CMAlarm, PT:= ParamTempoComAlarm, Q=>MesDataExd.MesData.MesAlarmCom) ;	 	


	FB_AlarmCodeManager(
		bAlarm1			:= MesDataExd.MesbAlarm, 					// HVAC Alarm Synthesis 
		bAlarm2			:= MesDataExd.MesData.MesAlarmCom,			// Communication Alarm #COM
		bAlarm3			:= WriteAlarm,					// Write Alarm 
		bAlarm4			:= FALSE,						//
		bAlarm5			:= False,                       //
		bAlarm6			:= False,                       //
		bAlarm7			:= False,                       //
		bAlarm8			:= False,                       //
		bAlarm9			:= FALSE,						//
		bAlarm10		:= False,                       //
		bAlarm11		:= False,                       //
		bAlarm12		:= False,                       //
		bAlarm13		:= False,                       //
		bAlarm14		:= FALSE,						//
		bAlarm15		:= False,                       //
		wAlarmCode		=>MesDataExd.MesData.MesAlarmCode);       
		                                                
                                                        
// WARNING CODE //
	FB_AlarmCodeManager
(
 		bAlarm1			:= MesWarningCom,						// Communication warning  #COM
		bAlarm2			:= False,                               //
		bAlarm3			:= False,                               //
		bAlarm4			:= False,                               //
		bAlarm5			:= False,                               //
		bAlarm6			:= False,                               //
		bAlarm7			:= False,                               //
		bAlarm8			:= False,                               //
		bAlarm9			:= False,                               //
		bAlarm10		:= False,                               //
		bAlarm11		:= False,                               //
		bAlarm12		:= FALSE,								//
		bAlarm13		:= False,                               //
		bAlarm14		:= False,                               //
		bAlarm15		:= False,                               //
		wAlarmCode		=>MesDataExd.MesData.MesWarningCode				
);   


// ALARM WORD EQUIPEMNT 
(*
	FB_AlarmCodeManager
(
		bAlarm0			:= ,// No active error                                           
 		bAlarm1			:= ,// Discharge Temperature high                                					   
		bAlarm2			:= ,// Internal thermostat detector working (49C)                                           
		bAlarm3			:= ,// Outdoor unit fail                                                                    
		bAlarm4			:= ,// Pressure low                                                                         
		bAlarm5			:= ,// Pressure high (High pressure probe working 63H)                                      
		bAlarm6			:= ,// Protection against freeze or battery high temperature                                
		bAlarm7			:= ,// Unknown Alarm 1                               
		bAlarm8			:= ,// Overheating protection                                                               
		bAlarm9			:= ,// High pressure error (ball valve closed)                                              
		bAlarm10		:= ,// Super heating anomaly due to low temp. of discharge. (TH4)                           
		bAlarm11		:= ,// Erroneous operation of drain pump                                                    
		bAlarm12		:= ,//  Unknown Alarm 2                   						
		bAlarm13		:= ,// Drain sensor anomaly (DS)                                                            
		bAlarm14		:= ,// Serial transmission error                                                            
		bAlarm15		:= ,// Compressor pause due to excess of current (initial block)                          
		wAlarmCode		=> MesDataExd.MesAlarm1			
);   

	FB_AlarmCodeManager
(
		bAlarm0			:= ,// Compressor pause due to excess of current (overload)
 		bAlarm1			:= ,// Phase detection opened                              				   
		bAlarm2			:= ,// Anti-phase detection                                                        
		bAlarm3			:= ,// Phase opened in phase L2 or connector 51CM opened                           
		bAlarm4			:= ,// Error in the anti-phase detector (electronic board)                         
		bAlarm5			:= ,// Connector 49L opened                                                        
		bAlarm6			:= ,// Cut due to over-current of compressor                                       
		bAlarm7			:= ,// Voltage anomaly                                                             
		bAlarm8			:= ,// Radiator panel temperature anomaly (TH8)                                    
		bAlarm9			:= ,// Ambient temperature probe anomaly (TH1), indoor unit                        
		bAlarm10		:= ,// Liquid probe anomaly (TH2)                                                  
		bAlarm11		:= ,// Cond/Evap probe anomaly (TH5)                                               
		bAlarm12		:= ,// Error detection in discharge temperature            					
		bAlarm13		:= ,// Outdoor probe error TH3                                                     
		bAlarm14		:= ,// Outdoor probe errorTH7                                                      
		bAlarm15		:= ,// Outdoor probe errorTH6                                                    
		wAlarmCode		=> MesDataExd.MesAlarm2			
);   

	FB_AlarmCodeManager
(
		bAlarm0			:= ,// Outdoor probe errorTH8                                                                                    
 		bAlarm1			:= ,// Connector 63L opened                                                                                      			   
		bAlarm2			:= ,// Current probe error                                                                                                             
		bAlarm3			:= ,// MNET duplicated address definition                                                                                              
		bAlarm4			:= ,// MNET Line transmission hardware error                                                                                           
		bAlarm5			:= ,// MNET BUS busy                                                                                                                   
		bAlarm6			:= ,// MNET Line transmission error                                                                                                    
		bAlarm7			:= ,// MNET transmission error                                                                                                         
		bAlarm8			:= ,// MNET without ack                                                                                                                
		bAlarm9			:= ,// MNET transmission error                                                                                                         
		bAlarm10		:= ,// MNET without response                                                                                                           
		bAlarm11		:= ,// AC’s remote command transmission error (reception error)                                                                        
		bAlarm12		:= ,// AC’s remote command transmission error (transmission error)                                               				
		bAlarm13		:= ,// Transmission error with the indoor/outdoor unit (reception error)                                                               
		bAlarm14		:= ,// Transmission error with the indoor/outdoor unit (transmission error)                                                            
		bAlarm15		:= ,// Error in inter-connection cable in the indoor/outdoor unit, indoor unit number deactivated (5 min or more)                   
		wAlarmCode		=> MesDataExd.MesAlarm3		
);   


	FB_AlarmCodeManager
(
		bAlarm0			:= ,// Error in inter-connection cable in the indoor/outdoor unit (cabling error, disconnection)
 		bAlarm1			:= ,// Initial timer deactivated                                                                	   
		bAlarm2			:= ,// Initializing                                                                        
		bAlarm3			:= ,//                                                                                                          
		bAlarm4			:= ,//                 
		bAlarm5			:= ,//                 
		bAlarm6			:= ,//                 
		bAlarm7			:= ,//                 
		bAlarm8			:= ,//                 
		bAlarm9			:= ,//                 
		bAlarm10		:= ,//                 
		bAlarm11		:= ,//                 
		bAlarm12		:= ,// 		
		bAlarm13		:= ,//                 
		bAlarm14		:= ,//                 
		bAlarm15		:= ,//              
		wAlarmCode		=> MesDataExd.MesAlarm4	
);  







*)
END_METHOD

METHOD M_CP : BOOL
VAR_INPUT
END_VAR


SUPER^.M_CP() ; 




Trig_Cmd_Read(CLK:=IN_CmdToggleRead);
Trig_Cmd_Write(CLK:=IN_CmdToggleWrite);
	
IF Trig_Cmd_Read.Q THEN
	IN_CmdToggleRead := FALSE;
	MesDataExd.MesData.MesCP_Read := NOT MesDataExd.MesData.MesCP_Read;
END_IF


IF Trig_Cmd_Write.Q THEN
	IN_CmdToggleWrite := FALSE;
	MesDataExd.MesData.MesCP_Write := NOT MesDataExd.MesData.MesCP_Write;
END_IF
END_METHOD

METHOD M_Evaluate : BOOL
VAR_INPUT
END_VAR


MesDataExd.MesAlarm1.0 := MesDataExd.MesErrorCode = 0;
MesDataExd.MesAlarm1.1 := MesDataExd.MesErrorCode = 1102;
MesDataExd.MesAlarm1.2 := MesDataExd.MesErrorCode = 1108;
MesDataExd.MesAlarm1.3 := MesDataExd.MesErrorCode = 1110;
MesDataExd.MesAlarm1.4 := MesDataExd.MesErrorCode = 1300;
MesDataExd.MesAlarm1.5 := MesDataExd.MesErrorCode = 1302;
MesDataExd.MesAlarm1.6 := MesDataExd.MesErrorCode = 1503;
MesDataExd.MesAlarm1.7 := MesDataExd.MesErrorCode = 1504;
MesDataExd.MesAlarm1.8 := MesDataExd.MesErrorCode = 1504;
MesDataExd.MesAlarm1.9 := MesDataExd.MesErrorCode = 1509;
MesDataExd.MesAlarm1.10:= MesDataExd.MesErrorCode = 1520;
MesDataExd.MesAlarm1.11:= MesDataExd.MesErrorCode = 2500;
MesDataExd.MesAlarm1.12:= MesDataExd.MesErrorCode = 2502;
MesDataExd.MesAlarm1.13:= MesDataExd.MesErrorCode = 2503;
MesDataExd.MesAlarm1.14:= MesDataExd.MesErrorCode = 4030;
MesDataExd.MesAlarm1.15:= MesDataExd.MesErrorCode = 4100;
MesDataExd.MesAlarm2.0 := MesDataExd.MesErrorCode = 4101;
MesDataExd.MesAlarm2.1 := MesDataExd.MesErrorCode = 4102;
MesDataExd.MesAlarm2.2 := MesDataExd.MesErrorCode = 4103;
MesDataExd.MesAlarm2.3 := MesDataExd.MesErrorCode = 4108;
MesDataExd.MesAlarm2.4 := MesDataExd.MesErrorCode = 4118;
MesDataExd.MesAlarm2.5 := MesDataExd.MesErrorCode = 4124;
MesDataExd.MesAlarm2.6 := MesDataExd.MesErrorCode = 4210;
MesDataExd.MesAlarm2.7 := MesDataExd.MesErrorCode = 4220;
MesDataExd.MesAlarm2.8 := MesDataExd.MesErrorCode = 4230;
MesDataExd.MesAlarm2.9 := MesDataExd.MesErrorCode = 5101;
MesDataExd.MesAlarm2.10:= MesDataExd.MesErrorCode = 5102;
MesDataExd.MesAlarm2.11:= MesDataExd.MesErrorCode = 5102;
MesDataExd.MesAlarm2.12:= MesDataExd.MesErrorCode = 5104;
MesDataExd.MesAlarm2.13:= MesDataExd.MesErrorCode = 5105;
MesDataExd.MesAlarm2.14:= MesDataExd.MesErrorCode = 5106;
MesDataExd.MesAlarm2.15:= MesDataExd.MesErrorCode = 5107;
MesDataExd.MesAlarm3.0 := MesDataExd.MesErrorCode = 5110;
MesDataExd.MesAlarm3.1 := MesDataExd.MesErrorCode = 5202;
MesDataExd.MesAlarm3.2 := MesDataExd.MesErrorCode = 5300;
MesDataExd.MesAlarm3.3 := MesDataExd.MesErrorCode = 6600;
MesDataExd.MesAlarm3.4 := MesDataExd.MesErrorCode = 6602;
MesDataExd.MesAlarm3.5 := MesDataExd.MesErrorCode = 6603;
MesDataExd.MesAlarm3.6 := MesDataExd.MesErrorCode = 6606;
MesDataExd.MesAlarm3.7 := MesDataExd.MesErrorCode = 6607;
MesDataExd.MesAlarm3.8 := MesDataExd.MesErrorCode = 6607;
MesDataExd.MesAlarm3.9 := MesDataExd.MesErrorCode = 6608;
MesDataExd.MesAlarm3.10:= MesDataExd.MesErrorCode = 6608;
MesDataExd.MesAlarm3.11:= MesDataExd.MesErrorCode = 6831;
MesDataExd.MesAlarm3.12:= MesDataExd.MesErrorCode = 6832;
MesDataExd.MesAlarm3.13:= MesDataExd.MesErrorCode = 6840;
MesDataExd.MesAlarm3.14:= MesDataExd.MesErrorCode = 6841;
MesDataExd.MesAlarm3.15:= MesDataExd.MesErrorCode = 6844;
MesDataExd.MesAlarm4.0 := MesDataExd.MesErrorCode = 6845;
MesDataExd.MesAlarm4.1 := MesDataExd.MesErrorCode = 6846;
MesDataExd.MesAlarm4.2 := MesDataExd.MesErrorCode = 65535;
END_METHOD

METHOD M_Read : BOOL
VAR
		MW 					: FB_MergeWordsToDint; 
	MesAlarm1: WORD;
	MesAlarm3: WORD;
	MesAlarm2: WORD;
	
	MesOn : REAL;
	MesData: INT;
END_VAR


IF MesDataExd.MesData.MesCP_Read  THEN	

	InputStructRead.InBuffer := ADR(MesBlock1_Temp);
	InputStructRead.InFunction := 4;
	InputStructRead.InQuantity := 97;
	InputStructRead.InStartAddr := 0;
	InputStructRead.InUnitID := ParamUnitID;
	InputStructRead.OutBusy := ADR(bReadBusy);
	InputStructRead.OutError := ADR(bReadError);
	InputStructRead.OutCompleted := ADR(bReadCompleted);
	
	
	MesDataExd.MesData.MesOn := MesBlock1_Temp[1] = 1;
	MesDataExd.MesMode := MesBlock1_Temp[2];
	MesDataExd.MesFanMode := MesBlock1_Temp[3];
	
	TRIG_Read(CLK := ClockRead);
	IF TRIG_Read.Q THEN	
		AX_ESS[ParamNumEss].ModbusRTU.M_AddAction_FIFO(InPriority := 2, InStruct := InputStructRead);
	END_IF
	
	MW(WORD_STRONG := MesBlock1_Temp[5], SIZE:= 1, Fix := 0, SIGNED := TRUE, VAR_OUT := MesDataExd.MesData.MesSetptTemp);
	MW(WORD_STRONG := MesBlock1_Temp[6], SIZE:= 1, Fix := 0, SIGNED := TRUE, VAR_OUT := MesDataExd.MesTempRoom);
	MW(WORD_STRONG := MesBlock1_Temp[10], SIZE:= 1, Fix := 0, SIGNED := TRUE, VAR_OUT := MesDataExd.MesData.MesWorkingHr);
	

	MesDataExd.MesbAlarm := MesBlock1_Temp[11] = 1;
	MesDataExd.MesErrorCode := MesBlock1_Temp[12] ;
	MW(WORD_STRONG := MesBlock1_Temp[24], SIZE:= 1, Fix := 0, SIGNED := TRUE, VAR_OUT := MesDataExd.MesTempRealSetpt);
END_IF
END_METHOD

METHOD M_Write : BOOL
VAR_INPUT
END_VAR
VAR
	
	WriteCmd1: BOOL;
	WriteCmd2: BOOL;

END_VAR
MesDataExd.IN_SetptTemp := MAX( ParamTempMin, MIN(ParamTempMax, IN_SetptTemp));

Trig_CmdStart(CLK := IN_CmdStart);
Trig_CmdStop(CLk := IN_CmdStop);

RS_StartStop(SET := Trig_CmdStop.Q, RESET1 := Trig_CmdStart.Q);

IF Trig_CmdStart.Q THEN
	IN_CmdStart := FALSE;
END_IF

IF Trig_CmdStop.Q THEN
	IN_CmdStop := FALSE;
END_IF

IF MesDataExd.MesData.MesCP_Write THEN
	// Setpoint 
	TRIG_Write(CLK := ClockWrite);
	

	InputStructWrite[1].InBuffer := ADR(WordToWrite1);
	InputStructWrite[1].InFunction := 6;
	InputStructWrite[1].InQuantity := 1;
	InputStructWrite[1].InStartAddr := 4;
	InputStructWrite[1].InUnitID := ParamUnitID;
	InputStructWrite[1].OutBusy := ADR(bWriteBusy[1]);
	InputStructWrite[1].OutError := ADR(bWriteError[1]);
	InputStructWrite[1].OutCompleted := ADR(bWriteCompleted[1]);
	
	WordToWrite1 := REAL_TO_WORD(MesDataExd.IN_SetptTemp);
	IF WordToWrite1 <> WordToWrite1_Old THEN
		WordToWrite1_Old := WordToWrite1;
		AX_ESS[ParamNumEss].ModbusRTU.M_AddAction_FIFO(InPriority := 2, InStruct := InputStructWrite[1]);
		
	END_IF

	// CmdStart/Stop
	InputStructWrite[2].InBuffer := ADR(WordToWrite2);          
	InputStructWrite[2].InFunction := 6;                        
	InputStructWrite[2].InQuantity := 1;                        
	InputStructWrite[2].InStartAddr := 0;                       
	InputStructWrite[2].InUnitID := ParamUnitID;                
	InputStructWrite[2].OutBusy := ADR(bWriteBusy[2]);          
	InputStructWrite[2].OutError := ADR(bWriteError[2]);        
	InputStructWrite[2].OutCompleted := ADR(bWriteCompleted[2]);
	
	WordToWrite2 := BOOL_TO_WORD(NOT RS_StartStop.Q1);
	IF WordToWrite2 <> WordToWrite2_Old THEN
		WordToWrite2_Old := WordToWrite2;
		AX_ESS[ParamNumEss].ModbusRTU.M_AddAction_FIFO(InPriority := 2, InStruct := InputStructWrite[2]);
		
	END_IF
END_IF
END_METHOD

END_FUNCTION_BLOCK

// ---- 01_Equipement_Library/HVAC/FB_HVAC_Base.TcPOU
FUNCTION_BLOCK FB_HVAC_Base
VAR_INPUT PERSISTENT
	ParamClockWriteTime						: TIME 		:= T#2S;	(* Modbus Writing Frequency                 *)
	ParamClockReadTime						: TIME 		:= T#1S;	(* Modbus Reading  Frequency                *)	


END_VAR

VAR_INPUT
		IN_CmdToggleRead						: BOOL;
    IN_CmdToggleWrite						: BOOL;
END_VAR

VAR

	//M_CP VARIABLES//
		Trig_Cmd_Read						: R_TRIG;                                                                                        
		Trig_Cmd_Write						: R_TRIG;                                                                                        

	
		TP1								: TP;
		TP2								: TP;
		TpUpdate						: TP;
		Trig_CmdStart					: R_TRIG;
		Trig_CmdReset					: R_TRIG;
		FTrig_CmdReset					: F_TRIG ; 
		Trig_CmdStop					: R_TRIG;
		WorkingHr						: TIME ; 
	
	///MesDataExd			AT%Q*		: HVAC;
	
		ClockWrite				AT%Q*		: BOOL;
		ClockRead				AT%Q*		: BOOL;
		
END_VAR
VAR_OUTPUT PERSISTENT
		OUT_State							: BOOL;
        OUT_WorkingHr						: TIME;                  			
END_VAR

METHOD M_AlarmManagement : BOOL
VAR_INPUT
END_VAR

VAR
	FB_AlarmCodeManager			: FB_AlarmCodeManager ;
END_VAR
END_METHOD

METHOD M_CP : BOOL
VAR_INPUT
END_VAR
END_METHOD

METHOD M_Evaluate : BOOL
VAR_INPUT
END_VAR
END_METHOD

METHOD M_Execute : BOOL
VAR_INPUT
END_VAR
TP1(IN:=NOT TP1.Q , PT:= ParamClockWriteTime);
ClockWrite 	:= TP1.Q ;
TP2(IN:=NOT TP2.Q , PT:= ParamClockReadTime);
ClockRead 	:= TP2.Q ;

TpUpdate(IN := NOT TpUpdate.Q, PT := T#5M);
	

	M_Evaluate();
	M_AlarmManagement();
	M_CP();
	M_Write();
	M_Read();
END_METHOD

METHOD M_Read : BOOL
VAR_INPUT
END_VAR
END_METHOD

METHOD M_Write : BOOL
VAR_INPUT
END_VAR
VAR
	WordToWrite		: WORD;
	AX_Addr			: ARRAY[1..3] OF UINT :=[1, 2, 3];
	
END_VAR
END_METHOD

END_FUNCTION_BLOCK

// ---- 01_Equipement_Library/HVAC/FB_HVAC_Standard.TcPOU
FUNCTION_BLOCK FB_HVAC_Standard EXTENDS FB_HVAC_Base
VAR_INPUT PERSISTENT
	{attribute 'OPC.UA.DA' := '1'} 
	ParamIpAddress							: STRING;
	{attribute 'OPC.UA.DA' := '1'} 
	ParamUnitID								: BYTE  := 1 ; 
	{attribute 'OPC.UA.DA' := '1'}                  
	ParamTcpPort							: UINT 	:= 502;
	ParamPriority							: UINT; 

	ParamTimeOut							: TIME 	:= T#2S;
	ParamMaintainPulse						: TIME 	:= T#2S;
END_VAR

VAR_INPUT
	IN_SetptTemp				AT%Q*		: REAL;
	IN_SetptHygro				AT%Q*		: REAL;
	IN_CmdStart								: BOOL;
	IN_CmdStop								: BOOL;
	IN_CmdReset_L							: BOOL;
		MesDataExd								: HVAC_Standard ; 
END_VAR

VAR

                                                                                 

		
	//M_READ VARIABLES//
		WriteSetpt							: FB_ModbusWriteSingleRegister;
		WriteCmd							: FB_ModbusWriteSingleCoil;
		ReadStatus							: FB_ModbusReadCoils;
		

		BlockToWrite			AT%Q*		: UINT;			
		TP_MaintainStart				: TP;
		R_TrigWriteCmd					: R_TRIG;
		F_TrigWriteCmd					: F_TRIG;

		R_TrigState						: R_TRIG;
		F_TrigState						: F_TRIG;
		TimeStart						: TIME;
		TimeNotStart					: TIME;
		
END_VAR

METHOD M_AlarmManagement : BOOL
VAR_INPUT
END_VAR

VAR
	FB_AlarmCodeManager			: FB_AlarmCodeManager ;
END_VAR
	FB_AlarmCodeManager(
		bAlarm1			:= FALSE, 	// CB of the battery charger is opened
		bAlarm2			:= FALSE,			// Main switch of tgbt is opened
		bAlarm3			:= False,	// No Voltage on the 48V TGBT
		bAlarm4			:= False,
		bAlarm5			:= False,
		bAlarm6			:= False,
		bAlarm7			:= False,
		bAlarm8			:= False,
		bAlarm9			:= False,
		bAlarm10		:= False,
		bAlarm11		:= False,
		bAlarm12		:= False,
		bAlarm13		:= False,
		bAlarm14		:= False,
		bAlarm15		:= False,
		wAlarmCode		=>MesDataExd.MesData.MesAlarmCode); 
		

// WARNING CODE //
	FB_AlarmCodeManager
(
 		bAlarm1			:= FALSE,
		bAlarm2			:= False,
		bAlarm3			:= False,
		bAlarm4			:= False,
		bAlarm5			:= False,
		bAlarm6			:= False,
		bAlarm7			:= False,
		bAlarm8			:= False,
		bAlarm9			:= False,
		bAlarm10		:= False,
		bAlarm11		:= False,
		bAlarm12		:= False,
		bAlarm13		:= False,
		bAlarm14		:= False,
		bAlarm15		:= False,
		wAlarmCode		=>MesDataExd.MesData.MesWarningCode					
);
END_METHOD

METHOD M_CP : BOOL
VAR_INPUT
END_VAR


SUPER^.M_CP() ; 




Trig_Cmd_Read(CLK:=IN_CmdToggleRead);
Trig_Cmd_Write(CLK:=IN_CmdToggleWrite);
	
IF Trig_Cmd_Read.Q THEN
	IN_CmdToggleRead := FALSE;
	MesDataExd.MesData.MesCP_Read := NOT MesDataExd.MesData.MesCP_Read;
END_IF


IF Trig_Cmd_Write.Q THEN
	IN_CmdToggleWrite := FALSE;
	MesDataExd.MesData.MesCP_Write := NOT MesDataExd.MesData.MesCP_Write;
END_IF
END_METHOD

METHOD M_Evaluate : BOOL
VAR_INPUT
END_VAR
END_METHOD

METHOD M_Read : BOOL
VAR_INPUT
END_VAR

IF MesDataExd.MesData.MesCP_Read  THEN	

